# B&R Automation Studio project Panasonic_LinkaPowerCP2_A2021055 (part 5)

```iecst
(*//P4 - Spodný stoper//*)

TYPE
	P4_SpodnyStoper_typ : 	STRUCT
		IN : P4_SpodnyStoper_IN_typ;
		OUT : P4_SpodnyStoper_OUT_typ;
		PAR : P4_SpodnyStoper_PAR_typ;
		STAV : P4_SpodnyStoper_STAV_typ;
		Automat : BOOL;
		Manual : BOOL;
		Reset : BOOL;
		KoniecCyklu : BOOL;
	END_STRUCT;
	P4_SpodnyStoper_IN_typ : 	STRUCT
		PritomnostPaletky : BOOL; (*IS4_15*)
		ZaplnenieDopravnika : BOOL; (*IS4_16*)
	END_STRUCT;
	P4_SpodnyStoper_OUT_typ : 	STRUCT
		ZasunStoper : BOOL; (*YV182_VT4*)
	END_STRUCT;
	P4_SpodnyStoper_PAR_typ : 	STRUCT
		New_Member : USINT;
	END_STRUCT;
	P4_SpodnyStoper_STAV_typ : 	STRUCT
		PoINIT : BOOL;
		PrebiehaVyvezeniePaletky : BOOL;
	END_STRUCT;
END_TYPE

(*//P4 - Funkčný test A//*)

TYPE
	P4_FunkcnyTestA_typ : 	STRUCT
		CMD : P4_FunkcnyTestA_CMD_typ;
		IN : P4_FunkcnyTestA_IN_typ;
		OUT : P4_FunkcnyTestA_OUT_typ;
		PAR : P4_FunkcnyTestA_PAR_typ;
		STAV : P4_FunkcnyTestA_STAV_typ;
		RFID_hlava : SickHeads;
		Automat : BOOL;
		Manual : BOOL;
		Reset : BOOL;
		KoniecCyklu : BOOL;
	END_STRUCT;
	P4_FunkcnyTestA_CMD_typ : 	STRUCT
		RR_ZatvorTester : BOOL;
		StartTestovania : BOOL;
		RR_VysunCentrovanie : BOOL;
		RR_VysunPruzenieKontaktov : BOOL;
		OpatovnyTest : BOOL;
	END_STRUCT;
	P4_FunkcnyTestA_IN_typ : 	STRUCT
		HorneKontakty_VYSUNUTE : BOOL; (*MS4_2*)
		HorneKontakty_ZASUNUTE : BOOL; (*MS4_3*)
		SpodneKontakty_VYSUNUTE : BOOL; (*MS4_7*)
		SpodneKontakty_ZASUNUTE : BOOL; (*MS4_6*)
		Centrovanie_VYSUNUTE : BOOL; (*MS4_5*)
		Centrovanie_ZASUNUTE : BOOL; (*MS4_4*)
		TypSpodnychKontaktov_4F : BOOL;
		TypSpodnychKontaktov_5F_5H : BOOL;
	END_STRUCT;
	P4_FunkcnyTestA_OUT_typ : 	STRUCT
		ZasunStoper : BOOL; (*YV170_VT4*)
		HorneKontakty_VYSUN : BOOL; (*YV193_VT4*)
		HorneKontakty_ZASUN : BOOL; (*YV192_VT4*)
		OdpruzHornychKontaktov_VYSUN : BOOL; (*YV194_VT4*)
		OdpruzHornychKontaktov_ZASUN : BOOL; (*YV195_VT4*)
		PritlakPowerCP_VYSUN : BOOL; (*YV196_VT4*)
		SpodneKontakty_VYSUN : BOOL; (*YV200_VT4*)
		SpodneKontakty_ZASUN : BOOL; (*YV199_VT4*)
		Centrovanie_VYSUN : BOOL; (*YV197_VT4*)
		Centrovanie_ZASUN : BOOL; (*YV198_VT4*)
		KontaktyTestera_VYSUN : BOOL;
	END_STRUCT;
	P4_FunkcnyTestA_PAR_typ : 	STRUCT
		CisloPaletky_STRING : STRING[2];
		CisloPortuKlienta : UINT;
	END_STRUCT;
	P4_FunkcnyTestA_STAV_typ : 	STRUCT
		PoINIT : BOOL;
		Vysledok_FV_Testu : STRING[2]; (*OK alebo NG*)
		PrebiehaVyvezeniePaletky : BOOL;
		Tester_ON : BOOL;
		TestovanieUkoncene : BOOL;
		TesterNeodpoveda : BOOL;
		RR_SekvenciaTestera_BUSY : BOOL;
		PaletkaOznacena_NG : BOOL;
	END_STRUCT;
END_TYPE

(*//P4 - Funkčný test B//*)

TYPE
	P4_FunkcnyTestB_typ : 	STRUCT
		CMD : P4_FunkcnyTestB_CMD_typ;
		IN : P4_FunkcnyTestB_IN_typ;
		OUT : P4_FunkcnyTestB_OUT_typ;
		PAR : P4_FunkcnyTestB_PAR_typ;
		STAV : P4_FunkcnyTestB_STAV_typ;
		RFID_hlava : SickHeads;
		Automat : BOOL;
		Manual : BOOL;
		Reset : BOOL;
		KoniecCyklu : BOOL;
	END_STRUCT;
	P4_FunkcnyTestB_CMD_typ : 	STRUCT
		RR_ZatvorTester : BOOL;
		StartTestovania : BOOL;
		RR_VysunCentrovanie : BOOL;
		RR_VysunPruzenieKontaktov : BOOL;
		OpatovnyTest : BOOL;
	END_STRUCT;
	P4_FunkcnyTestB_IN_typ : 	STRUCT
		HorneKontakty_VYSUNUTE : BOOL; (*MS4_8*)
		HorneKontakty_ZASUNUTE : BOOL; (*MS4_9*)
		SpodneKontakty_VYSUNUTE : BOOL; (*MS4_13*)
		SpodneKontakty_ZASUNUTE : BOOL; (*MS4_12*)
		Centrovanie_VYSUNUTE : BOOL; (*MS4_11*)
		Centrovanie_ZASUNUTE : BOOL; (*MS4_10*)
		TypSpodnychKontaktov_4F : BOOL;
		TypSpodnychKontaktov_5F_5H : BOOL;
	END_STRUCT;
	P4_FunkcnyTestB_OUT_typ : 	STRUCT
		ZasunStoper : BOOL; (*YV171_VT4*)
		HorneKontakty_VYSUN : BOOL; (*YV202_VT4*)
		HorneKontakty_ZASUN : BOOL; (*YV201_VT4*)
		OdpruzHornychKontaktov_VYSUN : BOOL; (*YV203_VT4*)
		OdpruzHornychKontaktov_ZASUN : BOOL; (*YV204_VT4*)
		PritlakPowerCP_VYSUN : BOOL; (*YV205_VT4*)
		SpodneKontakty_VYSUN : BOOL; (*YV209_VT4*)
		SpodneKontakty_ZASUN : BOOL; (*YV208_VT4*)
		Centrovanie_VYSUN : BOOL; (*YV206_VT4*)
		Centrovanie_ZASUN : BOOL; (*YV207_VT4*)
		KontaktyTestera_VYSUN : BOOL;
	END_STRUCT;
	P4_FunkcnyTestB_PAR_typ : 	STRUCT
		CisloPaletky_STRING : STRING[2];
		CisloPortuKlienta : UINT;
	END_STRUCT;
	P4_FunkcnyTestB_STAV_typ : 	STRUCT
		PoINIT : BOOL;
		Vysledok_FV_Testu : STRING[2]; (*OK alebo NG*)
		PrebiehaVyvezeniePaletky : BOOL;
		Tester_ON : BOOL;
		TestovanieUkoncene : BOOL;
		TesterNeodpoveda : BOOL;
		RR_SekvenciaTestera_BUSY : BOOL;
		PaletkaOznacena_NG : BOOL;
	END_STRUCT;
END_TYPE

(*//P4 - Zdvižka za Funkčným Testom A//*)

TYPE
	P4_ZdvizkaZaFunkcTestA_typ : 	STRUCT
		IN : P4_ZdvizkaZaFunkTestA_IN_typ;
		OUT : P4_ZdvizkaZaFunkTestA_OUT_typ;
		PAR : P4_ZdvizkaZaFunkTestA_PAR_typ;
		STAV : P4_ZdvizkaZaFunkTestA_STAV_typ;
		Automat : BOOL;
		Manual : BOOL;
		Reset : BOOL;
		KoniecCyklu : BOOL;
	END_STRUCT;
	P4_ZdvizkaZaFunkTestA_IN_typ : 	STRUCT
		PritomnostPaletky : BOOL; (*IS4_10*)
		PoziciaPaletky_OK : BOOL; (*IS4_9*)
		Zdvizka_HornaPoloha : BOOL; (*IS4_6*)
		Zdvizka_SpodnaPoloha : BOOL; (*IS4_5*)
		Zdvizka_StrednaPoloha : BOOL; (*IS4_7*)
		TlmicPaletky_ZASUNUTY : BOOL; (*MS4_1*)
	END_STRUCT;
	P4_ZdvizkaZaFunkTestA_OUT_typ : 	STRUCT
		Zdvizku_ZASUN : BOOL; (*YV173_VT4*)
		Zdvizku_VYSUN : BOOL; (*YV172_VT4*)
		TlmicPaletky_VYSUN : BOOL; (*YV175_VT4*)
		TlmicPaletky_ZASUN : BOOL; (*YV176_VT4*)
	END_STRUCT;
	P4_ZdvizkaZaFunkTestA_PAR_typ : 	STRUCT
		New_Member : USINT;
	END_STRUCT;
	P4_ZdvizkaZaFunkTestA_STAV_typ : 	STRUCT
		PoINIT : BOOL;
		PrebiehaVyvezeniePaletky : BOOL;
	END_STRUCT;
END_TYPE

(*//P4 - Zdvižka za Funkčným Testom B//*)

TYPE
	P4_ZdvizkaZaFunkcTestB_typ : 	STRUCT
		IN : P4_ZdvizkaZaFunkTestB_IN_typ;
		OUT : P4_ZdvizkaZaFunkTestB_OUT_typ;
		PAR : P4_ZdvizkaZaFunkTestB_PAR_typ;
		STAV : P4_ZdvizkaZaFunkTestB_STAV_typ;
		Automat : BOOL;
		Manual : BOOL;
		Reset : BOOL;
		KoniecCyklu : BOOL;
	END_STRUCT;
	P4_ZdvizkaZaFunkTestB_IN_typ : 	STRUCT
		PritomnostPaletky : BOOL; (*IS4_8*)
		Zdvizka_HornaPoloha : BOOL; (*IS4_11*)
		Zdvizka_StrednaPoloha : BOOL; (*IS4_12*)
	END_STRUCT;
	P4_ZdvizkaZaFunkTestB_OUT_typ : 	STRUCT
		Zdvizku_VYSUN : BOOL; (*YV177_VT4*)
		TlmicPaletky_VYSUN : BOOL; (*YV178_VT4*)
	END_STRUCT;
	P4_ZdvizkaZaFunkTestB_PAR_typ : 	STRUCT
		New_Member : USINT;
	END_STRUCT;
	P4_ZdvizkaZaFunkTestB_STAV_typ : 	STRUCT
		PoINIT : BOOL;
		PrebiehaVyvezeniePaletky : BOOL;
	END_STRUCT;
END_TYPE

(*//P4 - Etiketovanie//*)

TYPE
	P4_Etiketovacka_typ : 	STRUCT
		CMD : P4_Etiketovacka_CMD_typ;
		IN : P4_Etiketovacka_IN_typ;
		OUT : P4_Etiketovacka_OUT_typ;
		PAR : P4_Etiketovacka_PAR_typ;
		STAV : P4_Etiketovacka_STAV_typ;
		RFID_hlava : SickHeads;
		Automat : BOOL;
		Manual : BOOL;
		Reset : BOOL;
		KoniecCyklu : BOOL;
		ServoZdvihuAplikatora : ServoDriver;
	END_STRUCT;
	P4_Etiketovacka_CMD_typ : 	STRUCT
		RR_ZdvihAplikatora_HORE : BOOL;
		RR_ZdvihAplikatora_DOLE : BOOL;
		RR_NalepEtiketu : BOOL;
		RR_VysunCentrovanie : BOOL;
		RR_PrisavanieEtikety : BOOL;
	END_STRUCT;
	P4_Etiketovacka_IN_typ : 	STRUCT
		Centrovanie_VYSUNUTE : BOOL; (*IS4_13*)
		Centrovanie_ZASUNUTE : BOOL; (*IS4_14*)
		ZdvihAplikatora_HornyLimSnimac : BOOL; (*IS4_3*)
		ZdvihAplikatora_SpodnyLimSnimac : BOOL; (*IS4_4*)
		Aplikator_OtocenyVPRED : BOOL; (*MS4_15*)
		Aplikator_OtocenyVZAD : BOOL; (*MS4_14*)
		Aplikator_VYSUNUTY : BOOL; (*MS4_17*)
		Aplikator_ZASUNUTY : BOOL; (*MS4_16*)
		PrisavanieEtikety_Vakum_OK : BOOL; (*S4_6*)
		NapajanieTlaciarne_OK : BOOL;
		PritlakPowerCP_ZASUNUTY : BOOL; (*MS4_18*)
		PritlakPowerCP_VYSUNUTY_45F : BOOL; (*MS4_19*)
		PritlakPowerCP_VYSUNUTY_5H : BOOL; (*MS4_20*)
	END_STRUCT;
	P4_Etiketovacka_OUT_typ : 	STRUCT
		OfukEtikety_ON : BOOL; (*YV185_VT4*)
		PrisavanieEtikety_ON : BOOL; (*YV210_VT4*)
		PrisavanieEtikety_OFF : BOOL; (*YV211_VT4*)
		Aplikator_OtocVPRED : BOOL; (*YV187_VT4*)
		Aplikator_OtocVZAD : BOOL; (*YV186_VT4*)
		Aplikator_VYSUN : BOOL; (*YV188_VT4*)
		ZasunStoper : BOOL; (*YV179_VT4*)
		Centrovanie_VYSUN : BOOL; (*YV180_VT4*)
		Centrovanie_ZASUN : BOOL; (*YV181_VT4*)
		PritlakPowerCP_VYSUN : BOOL; (*YV191_VT4*)
	END_STRUCT;
	P4_Etiketovacka_PAR_typ : 	STRUCT
		IndexFotky : USINT;
		CisloPaletky_STRING : STRING[2];
		ZdvihAplikatora_JoggRychlost : REAL;
		CisloPaletky : USINT;
	END_STRUCT;
	P4_Etiketovacka_STAV_typ : 	STRUCT
		PoINIT : BOOL;
		PrebiehaVyvezeniePaletky : BOOL;
		PowerCP_ZhodaQRkodu_OK : BOOL;
		Etiketa_ZhodaQRkodu_OK : BOOL;
		RR_SekvenciaEtiketovania_BUSY : BOOL;
		VstupnaKamerovaKontrola : BOOL;
		VyrobaZacala : BOOL;
	END_STRUCT;
END_TYPE

(*//P4 - Výťah*)

TYPE
	P4_Vytah_typ : 	STRUCT
		CMD : P4_Vytah_CMD_typ;
		IN : P4_Vytah_IN_typ;
		OUT : P4_Vytah_OUT_typ;
		PAR : P4_Vytah_PAR_typ;
		STAV : P4_Vytah_STAV_typ;
		Banner : BannerIOlink;
		RFID_hlava : SickHeads;
		ServoZdvihuVytahu : ServoDriver;
		Automat : BOOL;
		Manual : BOOL;
		Reset : BOOL;
		KoniecCyklu : BOOL;
	END_STRUCT;
	P4_Vytah_CMD_typ : 	STRUCT
		RR_ChodDopravnika_VPRED : BOOL;
		RR_ChodDopravnika_VZAD : BOOL;
		Banner_LED_OFF : BOOL;
		RR_ZdvihVytahu_HORE : BOOL;
		RR_ZdvihVytahu_DOLE : BOOL;
	END_STRUCT;
	P4_Vytah_IN_typ : 	STRUCT
		PrechodDopravnika : BOOL; (*OS4_1*)
		ZdvihVytahu_HornyLimitnySnimac : BOOL; (*IS4_2*)
		ZdvihVytahu_SpodnyLimitnySnimac : BOOL; (*IS4_1*)
		StavRiadeniaDopravVytahu_READY : BOOL; (*M4_3*)
		TeplotaMotoraDopravVytahu_OK : BOOL; (*M4_3*)
	END_STRUCT;
	P4_Vytah_OUT_typ : 	STRUCT
		DopravnikChod_VPRED : BOOL; (*M4_3*)
		DopravnikChod_VZAD : BOOL; (*M4_3*)
		OsvetlenieVytahu_ON : BOOL;
	END_STRUCT;
	P4_Vytah_PAR_typ : 	STRUCT
		CisloPaletky_STRING : STRING[2];
		IndexFotky : USINT;
		Zdvih_JoggRychlost : REAL;
		RR_PrecitaneCisloPaletky : USINT;
		CisloPaletky : USINT;
	END_STRUCT;
	P4_Vytah_STAV_typ : 	STRUCT
		PrebiehaVyvezeniePaletky : BOOL;
		PoINIT : BOOL;
	END_STRUCT;
END_TYPE

(**************Skrutkovacky AtlasCopco***************************)

TYPE
	SkrutkovackaAtlasCopco_typ : 	STRUCT
		RESET_Poruchy : BOOL;
		RESET_Vysledkov : BOOL;
		START_Skrutkovania : BOOL;
		START_Utahovania : BOOL;
		Stav_VysledokPotvrdeny : BOOL;
		Stav_EmergencyStop : BOOL;
		Stav_READY_to_START : BOOL;
		Stav_MANUAL : BOOL;
		Stav_UtahovanieUkoncene : BOOL;
		Stav_VysledokUtahovania_OK : BOOL;
		Stav_VysledokUtahovania_NG : BOOL;
		Stav_SmerOtacania_VPRED : BOOL;
		Stav_BUSY : BOOL;
		Stav_ControlerSwitch_ON : BOOL;
		Stav_Station_READY : BOOL;
		Stav_NastrojPripojeny : BOOL;
		Stav_NastrojUtahuje : BOOL;
		Stav_CisloAktualnehoProgramu : USINT;
		CisloZadanehoProgramu : USINT;
		VyslednyReport : STRING[5];
	END_STRUCT;
END_TYPE

(**************Ateq Leakage Testery******************)

TYPE
	AteqTester_typ : 	STRUCT
		START_Testovania : BOOL;
		RESET_Vysledkov : BOOL;
		ZMEN_Program : BOOL;
		CitajParametreTestera : BOOL;
		Stav_RESET_DONE : BOOL;
		Stav_START_DONE : BOOL;
		Stav_ZmenaProgramu_DONE : BOOL;
		Stav_ERROR : BOOL;
		Stav_READY : BOOL;
		Stav_BUSY : BOOL;
		Stav_CitanieParametrov_OK : BOOL;
		Stav_CitanieParametrov_ERROR : BOOL;
		CisloZadanehoProgramu : UINT;
		CisloAktualnehoProgramu : UINT;
		VysledokTestovania_OK : BOOL;
		VysledokTestovania_NG : BOOL;
		Profinet_PLC_INPUTS : ARRAY[1..100]OF USINT;
		Profinet_PLC_OUTPUTS : ARRAY[1..100]OF USINT;
		ReadParameter_1 : UINT;
		ReadParameter_2 : UINT;
		ReadParameter_3 : UINT;
		ReadParameter_4 : UINT;
		ReadParameter_5 : DINT;
		PocetCitanychParametrov : USINT;
		IdentifikaciaParametra_1 : USINT;
		IdentifikaciaParametra_2 : USINT;
		IdentifikaciaParametra_3 : USINT;
		IdentifikaciaParametra_4 : USINT;
		CasPnenia : REAL;
		CasStabilizacie : REAL;
		TlakPlnenia : REAL;
		Tolerancia : REAL;
		TlakUniku : REAL;
	END_STRUCT;
END_TYPE

(***************Komunikácia zo serverom********************)

TYPE
	KOM_Server_typ : 	STRUCT
		CMD : KOM_Server_CMD_typ;
		INPUTS : KOM_Server_INPUTS_typ;
		OUTPUTS : KOM_Server_OUTPUTS_typ;
		STATUS : KOM_Server_STATUS_typ;
	END_STRUCT;
	KOM_Server_CMD_typ : 	STRUCT
		VyziadajStavPaletky_TYP1 : BOOL;
		PriradQRkodFiltra_TYP3 : BOOL;
		VyziadajCisloEtikety_TYP0 : BOOL;
		OdosliStavPaletky_TYP2 : BOOL;
		VyziadajStavPanatrace_TYP4 : BOOL;
	END_STRUCT;
	KOM_Server_INPUTS_typ : 	STRUCT
		TYP_Prikazu : STRING[1]; (*Typ*)
		CisloStanice : STRING[5]; (*Stanica*)
		CisloPaletky : STRING[10]; (*RFID paletky*)
		QRkodPowerCP : STRING[30]; (*Master number*)
		QRkodFiltra : STRING[30]; (*DPS1*)
		ID_Operatora : STRING[80]; (*Operator*)
		Report : STRING[4000]; (*DATA  - Oddelené bodkočiarkou*)
		StavPaletky : STRING[4]; (*PASS alebo FAIL*)
		IndexPaletky : USINT;
	END_STRUCT;
	KOM_Server_OUTPUTS_typ : 	STRUCT
		TYP_Prikazu : STRING[1]; (*Typ*)
		CisloStanice : STRING[5]; (*Stanica*)
		CisloPaletky : STRING[10]; (*RFID paletky*)
		QRkodPowerCP : STRING[30]; (*Master number*)
		QRkodFiltra : STRING[30]; (*DPS1*)
		ID_Operatora : STRING[8]; (*Operator*)
		CisloEtikety : STRING[31];
		DruhCinnostiNaPaletke : STRING[20]; (*PRD;ST1 alebo SMP;CAL;ST1 alebo RST;HVT;ST1*)
		PovolenieCinnostiNaPaletke : STRING[2]; (*OK alebo NG*)
	END_STRUCT;
	KOM_Server_STATUS_typ : 	STRUCT
		KomunikaciaUkoncena : BOOL;
		KomunikaciaError : BOOL;
		KOM_READY : BOOL;
	END_STRUCT;
END_TYPE

(***************Vysledné reporty***************************)

TYPE
	Reports_typ : 	STRUCT
		Kamery : ReportKamery_typ;
		Skrutkovacky : ReportSkrutkovacky_typ;
		Zvaranie : ReportZvarania_typ;
		LeakageTest : ReportLeakageTest_typ;
	END_STRUCT;
	ReportKamery_typ : 	STRUCT
		P1_CAM2_KontrolaPaletky : STRING[5]; (*Výtah*)
		P1_CAM4_KontrolaPinovDPS : STRING[5]; (*Výtah*)
		P1_CAM6_KontrolaPaletky : STRING[5]; (*Srobovanie*)
		P2_CAM1_KontrolaTesnenia : STRING[5];
		P2_CAM17_KontrolaPaletky : STRING[5]; (*Zakladanie tesnenia*)
		P2_CAM9_KontrolaPaletky : STRING[5]; (*Srobovanie matice*)
		P2_CAM10_KontrolaPaletky : STRING[5]; (*Srobovanie*)
		P2_CAM11_KontrolaZvaru : STRING[5]; (*Zvaranie*)
		P2_CAM11_KontrolaPowerCP : STRING[5]; (*Zvaranie*)
		P2_CAM12_KontrolaPaletky : STRING[5];
		P3_CAM13_KontrolaPaletky : STRING[5]; (*Srobovanie*)
		P4_CAM15_KontrolaPaletky : STRING[5]; (*Etiketovačka*)
		P4_CAM16_KontrolaPaletky : STRING[5]; (*Výtah*)
	END_STRUCT;
	ReportSkrutkovacky_typ : 	STRUCT
		Moment_ToleranciaMAX : ReportSrobov_MomentTolerMAX_typ;
		Moment_ToleranciaMIN : ReportSrobov_MomentTolerMIN_typ;
		Moment_NameranaHodnota : ReportSrobov_NameranyMoment_typ;
		Uhol_ToleranciaMAX : ReportSrobov_UholTolerMAX_typ;
		Uhol_ToleranciaMIN : ReportSrobov_UholTolerMIN_typ;
		Uhol_NameranaHodnota : ReportSrobov_NameranyUhol_typ;
		VyskaSkrutkovania : ReportSrobov_VyskaSkrutkov_typ;
		CasSkrutkovania : ReportSrobov_CasSkrutkov_typ;
		VyslednyReport : ReportSrobov_VyslednyReport_typ;
	END_STRUCT;
	ReportZvarania_typ : 	STRUCT
		Vyska : ReportZvarania_Vyska_typ;
		Moment : ReportZvarania_Moment_typ;
		Frekvencia : STRING[10];
		VyslednyReport : STRING[5];
	END_STRUCT;
	ReportZvarania_Vyska_typ : 	STRUCT
		LavyZvar : STRING[10];
		PravyZvar : STRING[10];
	END_STRUCT;
	ReportZvarania_Moment_typ : 	STRUCT
		LavyZvar : STRING[4];
		PravyZvar : STRING[4];
	END_STRUCT;
	ReportSrobov_MomentTolerMAX_typ : 	STRUCT
		P1_LavaSkrutkaK30 : STRING[10];
		P1_PravaSkrutkaK30 : STRING[10];
		P1_ZadnaSkrutkaM4 : STRING[10];
		P1_PrednaSkrutkaM4 : STRING[10];
		P1_SkrutkaDPS_M4 : STRING[10];
		P1_LavaSkrutkaM5 : STRING[10];
		P1_PravaSkrutkaM5 : STRING[10];
		P1_StrednaSkrutkaM5 : STRING[10];
		P2_MaticaM4 : STRING[10];
		P2_LavaSkrutkaM6 : STRING[10];
		P2_PravaSkrutkaM6 : STRING[10];
		P2_LavaSkrutkaM4 : STRING[10];
		P2_PravaSkrutkaM4 : STRING[10];
		P2_LavaSkrutkaM5 : STRING[10];
		P2_PravaSkrutkaM5 : STRING[10];
		P2_StrednaSkrutkaM4 : STRING[10];
		P3_SkrutkaK40 : STRING[10];
		P3_SkrutkaM5 : STRING[10];
	END_STRUCT;
	ReportSrobov_MomentTolerMIN_typ : 	STRUCT
		P1_LavaSkrutkaK30 : STRING[10];
		P1_PravaSkrutkaK30 : STRING[10];
		P1_ZadnaSkrutkaM4 : STRING[10];
		P1_PrednaSkrutkaM4 : STRING[10];
		P1_SkrutkaDPS_M4 : STRING[10];
		P1_LavaSkrutkaM5 : STRING[10];
		P1_PravaSkrutkaM5 : STRING[10];
		P1_StrednaSkrutkaM5 : STRING[10];
		P2_MaticaM4 : STRING[10];
		P2_LavaSkrutkaM6 : STRING[10];
		P2_PravaSkrutkaM6 : STRING[10];
		P2_LavaSkrutkaM4 : STRING[10];
		P2_PravaSkrutkaM4 : STRING[10];
		P2_LavaSkrutkaM5 : STRING[10];
		P2_PravaSkrutkaM5 : STRING[10];
		P2_StrednaSkrutkaM4 : STRING[10];
		P3_SkrutkaK40 : STRING[10];
		P3_SkrutkaM5 : STRING[10];
	END_STRUCT;
	ReportSrobov_NameranyMoment_typ : 	STRUCT
		P1_LavaSkrutkaK30 : STRING[10];
		P1_PravaSkrutkaK30 : STRING[10];
		P1_ZadnaSkrutkaM4 : STRING[10];
		P1_PrednaSkrutkaM4 : STRING[10];
		P1_SkrutkaDPS_M4 : STRING[10];
		P1_LavaSkrutkaM5 : STRING[10];
		P1_PravaSkrutkaM5 : STRING[10];
		P1_StrednaSkrutkaM5 : STRING[10];
		P2_MaticaM4 : STRING[10];
		P2_LavaSkrutkaM6 : STRING[10];
		P2_PravaSkrutkaM6 : STRING[10];
		P2_LavaSkrutkaM4 : STRING[10];
		P2_PravaSkrutkaM4 : STRING[10];
		P2_LavaSkrutkaM5 : STRING[10];
		P2_PravaSkrutkaM5 : STRING[10];
		P2_StrednaSkrutkaM4 : STRING[10];
		P3_SkrutkaK40 : STRING[10];
		P3_SkrutkaM5 : STRING[10];
	END_STRUCT;
	ReportSrobov_UholTolerMAX_typ : 	STRUCT
		P1_LavaSkrutkaK30 : STRING[10];
		P1_PravaSkrutkaK30 : STRING[10];
		P1_ZadnaSkrutkaM4 : STRING[10];
		P1_PrednaSkrutkaM4 : STRING[10];
		P1_SkrutkaDPS_M4 : STRING[10];
		P1_LavaSkrutkaM5 : STRING[10];
		P1_PravaSkrutkaM5 : STRING[10];
		P1_StrednaSkrutkaM5 : STRING[10];
		P2_MaticaM4 : STRING[10];
		P2_LavaSkrutkaM6 : STRING[10];
		P2_PravaSkrutkaM6 : STRING[10];
		P2_LavaSkrutkaM4 : STRING[10];
		P2_PravaSkrutkaM4 : STRING[10];
		P2_LavaSkrutkaM5 : STRING[10];
		P2_PravaSkrutkaM5 : STRING[10];
		P2_StrednaSkrutkaM4 : STRING[10];
		P3_SkrutkaK40 : STRING[10];
		P3_SkrutkaM5 : STRING[10];
	END_STRUCT;
	ReportSrobov_UholTolerMIN_typ : 	STRUCT
		P1_LavaSkrutkaK30 : STRING[10];
		P1_PravaSkrutkaK30 : STRING[10];
		P1_ZadnaSkrutkaM4 : STRING[10];
		P1_PrednaSkrutkaM4 : STRING[10];
		P1_SkrutkaDPS_M4 : STRING[10];
		P1_LavaSkrutkaM5 : STRING[10];
		P1_PravaSkrutkaM5 : STRING[10];
		P1_StrednaSkrutkaM5 : STRING[10];
		P2_MaticaM4 : STRING[10];
		P2_LavaSkrutkaM6 : STRING[10];
		P2_PravaSkrutkaM6 : STRING[10];
		P2_LavaSkrutkaM4 : STRING[10];
		P2_PravaSkrutkaM4 : STRING[10];
		P2_LavaSkrutkaM5 : STRING[10];
		P2_PravaSkrutkaM5 : STRING[10];
		P2_StrednaSkrutkaM4 : STRING[10];
		P3_SkrutkaK40 : STRING[10];
		P3_SkrutkaM5 : STRING[10];
	END_STRUCT;
	ReportSrobov_NameranyUhol_typ : 	STRUCT
		P1_LavaSkrutkaK30 : STRING[10];
		P1_PravaSkrutkaK30 : STRING[10];
		P1_ZadnaSkrutkaM4 : STRING[10];
		P1_PrednaSkrutkaM4 : STRING[10];
		P1_SkrutkaDPS_M4 : STRING[10];
		P1_LavaSkrutkaM5 : STRING[10];
		P1_PravaSkrutkaM5 : STRING[10];
		P1_StrednaSkrutkaM5 : STRING[10];
		P2_MaticaM4 : STRING[10];
		P2_LavaSkrutkaM6 : STRING[10];
		P2_PravaSkrutkaM6 : STRING[10];
		P2_LavaSkrutkaM4 : STRING[10];
		P2_PravaSkrutkaM4 : STRING[10];
		P2_LavaSkrutkaM5 : STRING[10];
		P2_PravaSkrutkaM5 : STRING[10];
		P2_StrednaSkrutkaM4 : STRING[10];
		P3_SkrutkaK40 : STRING[10];
		P3_SkrutkaM5 : STRING[10];
	END_STRUCT;
	ReportSrobov_VyskaSkrutkov_typ : 	STRUCT
		P1_LavaSkrutkaK30 : STRING[10];
		P1_PravaSkrutkaK30 : STRING[10];
		P1_ZadnaSkrutkaM4 : STRING[10];
		P1_PrednaSkrutkaM4 : STRING[10];
		P1_SkrutkaDPS_M4 : STRING[10];
		P1_LavaSkrutkaM5 : STRING[10];
		P1_PravaSkrutkaM5 : STRING[10];
		P1_StrednaSkrutkaM5 : STRING[10];
		P2_MaticaM4 : STRING[10];
		P2_LavaSkrutkaM6 : STRING[10];
		P2_PravaSkrutkaM6 : STRING[10];
		P2_LavaSkrutkaM4 : STRING[10];
		P2_PravaSkrutkaM4 : STRING[10];
		P2_LavaSkrutkaM5 : STRING[10];
		P2_PravaSkrutkaM5 : STRING[10];
		P2_StrednaSkrutkaM4 : STRING[10];
		P3_SkrutkaK40 : STRING[10];
		P3_SkrutkaM5 : STRING[10];
	END_STRUCT;
	ReportSrobov_CasSkrutkov_typ : 	STRUCT
		P1_LavaSkrutkaK30 : STRING[10];
		P1_PravaSkrutkaK30 : STRING[10];
		P1_ZadnaSkrutkaM4 : STRING[10];
		P1_PrednaSkrutkaM4 : STRING[10];
		P1_SkrutkaDPS_M4 : STRING[10];
		P1_LavaSkrutkaM5 : STRING[10];
		P1_PravaSkrutkaM5 : STRING[10];
		P1_StrednaSkrutkaM5 : STRING[10];
		P2_MaticaM4 : STRING[10];
		P2_LavaSkrutkaM6 : STRING[10];
		P2_PravaSkrutkaM6 : STRING[10];
		P2_LavaSkrutkaM4 : STRING[10];
		P2_PravaSkrutkaM4 : STRING[10];
		P2_LavaSkrutkaM5 : STRING[10];
		P2_PravaSkrutkaM5 : STRING[10];
		P2_StrednaSkrutkaM4 : STRING[10];
		P3_SkrutkaK40 : STRING[10];
		P3_SkrutkaM5 : STRING[10];
	END_STRUCT;
	ReportSrobov_VyslednyReport_typ : 	STRUCT
		P1_LavaSkrutkaK30 : STRING[5];
		P1_PravaSkrutkaK30 : STRING[5];
		P1_ZadnaSkrutkaM4 : STRING[5];
		P1_PrednaSkrutkaM4 : STRING[5];
		P1_SkrutkaDPS_M4 : STRING[5];
		P1_LavaSkrutkaM5 : STRING[5];
		P1_PravaSkrutkaM5 : STRING[5];
		P1_StrednaSkrutkaM5 : STRING[5];
		P2_MaticaM4 : STRING[5];
		P2_LavaSkrutkaM6 : STRING[5];
		P2_PravaSkrutkaM6 : STRING[5];
		P2_LavaSkrutkaM4 : STRING[5];
		P2_PravaSkrutkaM4 : STRING[5];
		P2_LavaSkrutkaM5 : STRING[5];
		P2_PravaSkrutkaM5 : STRING[5];
		P2_StrednaSkrutkaM4 : STRING[5];
		P3_SkrutkaK40 : STRING[5];
		P3_SkrutkaM5 : STRING[5];
	END_STRUCT;
	ReportLeakageTest_typ : 	STRUCT
		CasPlnenia : RepLeakTest_CasPlnenia_typ;
		CasStabilizacie : RepLeakTest_CasStabilizacie_typ;
		TlakPlnenia : RepLeakTest_TlakPlnenia_typ;
		TlakPritlaku : RepLeakTest_TlakPritlaku_typ;
		ToleranciaPritlaku_MIN : RepLeakTest_TolPritlakuMIN_typ;
		ToleranciaPritlaku_MAX : RepLeakTest_TolPritlakuMAX_typ;
		ToleranciaTlakUniku_MIN : RepLeakTest_TolTlakUnikuMIN_typ;
		ToleranciaTlakUniku_MAX : RepLeakTest_TolTlakUnikuMAX_typ;
		TlakUniku : RepLeakTest_TlakUniku_typ;
		Tolerancia : RepLeakTest_Tolerancia_typ;
		VyslednyReport : RepLeakTest_VyslednyReport_typ;
	END_STRUCT;
	RepLeakTest_CasPlnenia_typ : 	STRUCT
		StanicaA : STRING[10];
		StanicaB : STRING[10];
	END_STRUCT;
	RepLeakTest_CasStabilizacie_typ : 	STRUCT
		StanicaA : STRING[10];
		StanicaB : STRING[10];
	END_STRUCT;
	RepLeakTest_TlakPlnenia_typ : 	STRUCT
		StanicaA : STRING[10];
		StanicaB : STRING[10];
	END_STRUCT;
	RepLeakTest_TlakPritlaku_typ : 	STRUCT
		StanicaA : STRING[10];
		StanicaB : STRING[10];
	END_STRUCT;
	RepLeakTest_TolPritlakuMIN_typ : 	STRUCT
		StanicaA : STRING[10];
		StanicaB : STRING[10];
	END_STRUCT;
	RepLeakTest_TolPritlakuMAX_typ : 	STRUCT
		StanicaA : STRING[10];
		StanicaB : STRING[10];
	END_STRUCT;
	RepLeakTest_TlakUniku_typ : 	STRUCT
		StanicaA : STRING[10];
		StanicaB : STRING[10];
	END_STRUCT;
	RepLeakTest_TolTlakUnikuMIN_typ : 	STRUCT
		StanicaA : STRING[10];
		StanicaB : STRING[10];
	END_STRUCT;
	RepLeakTest_TolTlakUnikuMAX_typ : 	STRUCT
		StanicaA : STRING[10];
		StanicaB : STRING[10];
	END_STRUCT;
	RepLeakTest_Tolerancia_typ : 	STRUCT
		StanicaA : STRING[10];
		StanicaB : STRING[10];
	END_STRUCT;
	RepLeakTest_VyslednyReport_typ : 	STRUCT
		StanicaA : STRING[5];
		StanicaB : STRING[5];
	END_STRUCT;
END_TYPE

(****************Kamerove kontroly**************************)

TYPE
	CAM1_typ : 	STRUCT  (*P2_ST1_ZaklTesnenia - Kontrola tesnenia a QR kódu Power CP //CAM4//*)
		CMD : CAM1_Commands_typ;
		PAR : CAM1_Parametre_typ;
		STAV : CAM1_Status_typ;
		RESULT : CAM1_Results_typ;
		Profinet_PLC_INPUTS : ARRAY[0..100]OF USINT;
		Profinet_PLC_OUTPUTS : ARRAY[0..3]OF USINT;
	END_STRUCT;
	CAM1_Commands_typ : 	STRUCT
		Triger : BOOL;
		OdosliFotku : BOOL;
		VymazFotku : BOOL;
	END_STRUCT;
	CAM1_Parametre_typ : 	STRUCT
		ResultFotky : STRING[5];
	END_STRUCT;
	CAM1_Status_typ : 	STRUCT
		BUSY : BOOL;
		SWITCH : BOOL;
		READY : BOOL;
		OLD_SWITCH : BOOL;
		Results_READY : BOOL;
		Command_READY : BOOL;
		Command_ERROR : BOOL;
		Command_AKCEPTOVANY : BOOL;
		RunCounter : UINT;
		OldRunCounter : UINT;
		RunCounter_Byte0 : USINT;
		RunCounter_Byte1 : USINT;
	END_STRUCT;
	CAM1_Results_typ : 	STRUCT
		ZalozenieTesnenia_OK : BOOL;
		NepritomnostTesnenia : BOOL;
	END_STRUCT;
	CAM2_typ : 	STRUCT  (*P1_ST1_Vytah - kontrola kusov na paletke //CAM1//*)
		CMD : CAM2_Commands_typ;
		PAR : CAM2_Parametre_typ;
		STAV : CAM2_Status_typ;
		RESULT : CAM2_Results_typ;
		Profinet_PLC_INPUTS : ARRAY[0..100]OF USINT;
		Profinet_PLC_OUTPUTS : ARRAY[0..3]OF USINT;
	END_STRUCT;
	CAM2_Commands_typ : 	STRUCT
		Triger : BOOL;
		OdosliFotku : BOOL;
		VymazFotku : BOOL;
	END_STRUCT;
	CAM2_Parametre_typ : 	STRUCT
		ResultFotky : STRING[5];
	END_STRUCT;
	CAM2_Status_typ : 	STRUCT
		READY : BOOL;
		BUSY : BOOL;
		SWITCH : BOOL;
		OLD_SWITCH : BOOL;
		Results_READY : BOOL;
		Command_READY : BOOL;
		Command_ERROR : BOOL;
		Command_AKCEPTOVANY : BOOL;
		RunCounter : UINT;
		OldRunCounter : UINT;
		RunCounter_Byte0 : USINT;
		RunCounter_Byte1 : USINT;
	END_STRUCT;
	CAM2_Results_typ : 	STRUCT
		Paletka : CAM2_Paletka_typ;
		PowerCP : CAM2_PowerCP_typ;
	END_STRUCT;
	CAM2_PowerCP_typ : 	STRUCT
		New_Member : USINT;
	END_STRUCT;
	CAM2_Paletka_typ : 	STRUCT
		Pritom_PowerCP_5F : BOOL;
		Pritom_PowerCP_4F : BOOL;
		Pritom_PowerCP_5H : BOOL;
		Pritomn_Skeletonu_5H : BOOL;
		Pritomn_Skeletonu_4F5F : BOOL;
		Pritom_Busbarov_Spodne_5H : BOOL;
		Pritom_Busbaru_Spodny_5F : BOOL;
		Pritom_Busbaru_Spodny_4F : BOOL;
		Pritom_DPS_4F5F : BOOL;
		Pritom_Foamu_Lavy_4F5F : BOOL;
		Pritom_Foamu_Pravy_4F5F : BOOL;
	END_STRUCT;
	CAM3_typ : 	STRUCT  (*P1_ST1_Vytah - kontrola QR kódu DPS //Smart kamera//*)
		CMD : CAM3_Commands_typ;
		PAR : CAM3_Parametre_typ;
		STAV : CAM3_Status_typ;
		RESULT : CAM3_Results_typ;
		Profinet_QRkod_Znaky : ARRAY[0..31]OF USINT;
		Profinet_PLC_INPUTS : ARRAY[0..100]OF USINT;
		Profinet_PLC_OUTPUTS : ARRAY[0..3]OF USINT;
	END_STRUCT;
	CAM3_Commands_typ : 	STRUCT
		Triger : BOOL;
		OdosliFotku : BOOL;
		VymazFotku : BOOL;
	END_STRUCT;
	CAM3_Parametre_typ : 	STRUCT
		ResultFotky : STRING[5];
	END_STRUCT;
	CAM3_Status_typ : 	STRUCT
		BUSY : BOOL;
		SWITCH : BOOL;
		READY : BOOL;
		OLD_SWITCH : BOOL;
		Results_READY : BOOL;
		RunCounter : UINT;
		OldRunCounter : UINT;
		RunCounter_Byte0 : USINT;
		RunCounter_Byte1 : USINT;
	END_STRUCT;
	CAM3_Results_typ : 	STRUCT
		Paletka : CAM3_Paletka_typ;
		PowerCP : CAM3_PowerCP_typ;
	END_STRUCT;
	CAM3_PowerCP_typ : 	STRUCT
		New_Member : USINT;
	END_STRUCT;
	CAM3_Paletka_typ : 	STRUCT
		CitanieQRkodu_DPS_OK : BOOL;
		PrecitanyQRkod_DPS : STRING[32];
	END_STRUCT;
	CAM4_typ : 	STRUCT  (*P1_ST1_Vytah - kontrola klipov krytu DPS //CAM2//*)
		CMD : CAM4_Commands_typ;
		PAR : CAM4_Parametre_typ;
		STAV : CAM4_Status_typ;
		RESULT : CAM4_Results_typ;
		Profinet_PLC_INPUTS : ARRAY[0..100]OF USINT;
		Profinet_PLC_OUTPUTS : ARRAY[0..3]OF USINT;
	END_STRUCT;
	CAM4_Commands_typ : 	STRUCT
		Triger : BOOL;
		OdosliFotku : BOOL;
		VymazFotku : BOOL;
	END_STRUCT;
	CAM4_Parametre_typ : 	STRUCT
		ResultFotky : STRING[5];
	END_STRUCT;
	CAM4_Status_typ : 	STRUCT
		READY : BOOL;
		BUSY : BOOL;
		SWITCH : BOOL;
		OLD_SWITCH : BOOL;
		Results_READY : BOOL;
		Command_READY : BOOL;
		Command_ERROR : BOOL;
		Command_AKCEPTOVANY : BOOL;
		RunCounter : UINT;
		OldRunCounter : UINT;
		RunCounter_Byte0 : USINT;
		RunCounter_Byte1 : USINT;
	END_STRUCT;
	CAM4_Results_typ : 	STRUCT
		Paletka : CAM4_Paletka_typ;
		PowerCP : CAM4_PowerCP_typ;
	END_STRUCT;
	CAM4_PowerCP_typ : 	STRUCT
		New_Member : USINT;
	END_STRUCT;
	CAM4_Paletka_typ : 	STRUCT
		Pritomn_Pinu1_KrytDPS_4F5F : BOOL;
		Pritomn_Pinu2_KrytDPS_4F5F : BOOL;
		Pritomn_Pinu3_KrytDPS_4F5F : BOOL;
		Pritomn_Pinu4_KrytDPS_4F5F : BOOL;
		Pritomn_Pinu5_KrytDPS_4F5F : BOOL;
		Pritomn_Pinu6_KrytDPS_4F5F : BOOL;
		Pritom_DPS_4F5F : BOOL;
	END_STRUCT;
	CAM5_typ : 	STRUCT  (*P1_ST1_Vytah - kontrola QR kódu PowerCP//Smart kamera//*)
		CMD : CAM5_Commands_typ;
		PAR : CAM5_Parametre_typ;
		STAV : CAM5_Status_typ;
		RESULT : CAM5_Results_typ;
		Profinet_QRkod_Znaky : ARRAY[0..31]OF USINT;
		Profinet_PLC_INPUTS : ARRAY[0..100]OF USINT;
		Profinet_PLC_OUTPUTS : ARRAY[0..3]OF USINT;
	END_STRUCT;
	CAM5_Commands_typ : 	STRUCT
		Triger : BOOL;
		OdosliFotku : BOOL;
		VymazFotku : BOOL;
	END_STRUCT;
	CAM5_Parametre_typ : 	STRUCT
		ResultFotky : STRING[5];
	END_STRUCT;
	CAM5_Status_typ : 	STRUCT
		BUSY : BOOL;
		SWITCH : BOOL;
		READY : BOOL;
		OLD_SWITCH : BOOL;
		Results_READY : BOOL;
		RunCounter : UINT;
		OldRunCounter : UINT;
		RunCounter_Byte0 : USINT;
		RunCounter_Byte1 : USINT;
	END_STRUCT;
	CAM5_Results_typ : 	STRUCT
		Paletka : CAM5_Paletka_typ;
		PowerCP : CAM5_PowerCP_typ;
	END_STRUCT;
	CAM5_PowerCP_typ : 	STRUCT
		CitanieQRkodu_PowerCP_OK : BOOL;
		PrecitanyQRkod_PowerCP : STRING[32];
	END_STRUCT;
	CAM5_Paletka_typ : 	STRUCT
		New_Member : USINT;
	END_STRUCT;
	CAM6_typ : 	STRUCT  (*P1_ST2_StoperSkrutkovania - Kontrola paletky //CAM3//*)
		CMD : CAM6_Commands_typ;
		PAR : CAM6_Parametre_typ;
		STAV : CAM6_Status_typ;
		RESULT : CAM6_Results_typ;
		Profinet_PLC_INPUTS : ARRAY[0..100]OF USINT;
		Profinet_PLC_OUTPUTS : ARRAY[0..3]OF USINT;
	END_STRUCT;
	CAM6_Commands_typ : 	STRUCT
		Triger : BOOL;
		OdosliFotku : BOOL;
		VymazFotku : BOOL;
	END_STRUCT;
	CAM6_Parametre_typ : 	STRUCT
		ResultFotky : STRING[5];
	END_STRUCT;
	CAM6_Status_typ : 	STRUCT
		READY : BOOL;
		BUSY : BOOL;
		SWITCH : BOOL;
		OLD_SWITCH : BOOL;
		Results_READY : BOOL;
		Command_READY : BOOL;
		Command_ERROR : BOOL;
		Command_AKCEPTOVANY : BOOL;
		RunCounter : UINT;
		OldRunCounter : UINT;
		RunCounter_Byte0 : USINT;
		RunCounter_Byte1 : USINT;
	END_STRUCT;
	CAM6_Results_typ : 	STRUCT
		Paletka : CAM6_Paletka_typ;
		PowerCP : CAM6_PowerCP_typ;
	END_STRUCT;
	CAM6_PowerCP_typ : 	STRUCT
		Nepritom_LavyFoam_4F5F : BOOL;
		Nepritom_PravyFoam_4F5F : BOOL;
		Pritom_LavejSkrutkyK30 : BOOL;
		Pritom_PravejSkrutkyK30 : BOOL;
	END_STRUCT;
	CAM6_Paletka_typ : 	STRUCT
		Pritom_PowerCP_5H : BOOL;
		Pritom_PowerCP_4F : BOOL;
		Pritom_PowerCP_5F : BOOL;
		Pritom_DPS_45F : BOOL;
		Pritom_SpodnychBusbarov_5H : BOOL;
		Pritom_SpodnyBusbar_5F : BOOL;
		Pritom_SpodnyBusbar_4F : BOOL;
		Pritom_LavyFoam_4F5F : BOOL;
		Pritom_PravyFoam_4F5F : BOOL;
	END_STRUCT;
	CAM7_typ : 	STRUCT  (*P2_ST1_StoperZaklTesnenia - Kontrola Power CP a QR kódu filtra //CAM5//*)
		CMD : CAM7_Commands_typ;
		PAR : CAM7_Parametre_typ;
		STAV : CAM7_Status_typ;
		RESULT : CAM7_Results_typ;
		Profinet_QRkod_Znaky : ARRAY[0..31]OF USINT;
		Profinet_PLC_INPUTS : ARRAY[0..100]OF USINT;
		Profinet_PLC_OUTPUTS : ARRAY[0..3]OF USINT;
	END_STRUCT;
	CAM7_Commands_typ : 	STRUCT
		Triger : BOOL;
		OdosliFotku : BOOL;
		VymazFotku : BOOL;
	END_STRUCT;
	CAM7_Parametre_typ : 	STRUCT
		ResultFotky : STRING[5];
	END_STRUCT;
	CAM7_Status_typ : 	STRUCT
		BUSY : BOOL;
		SWITCH : BOOL;
		READY : BOOL;
		OLD_SWITCH : BOOL;
		Results_READY : BOOL;
		Command_READY : BOOL;
		Command_ERROR : BOOL;
		Command_AKCEPTOVANY : BOOL;
		RunCounter : UINT;
		OldRunCounter : UINT;
		RunCounter_Byte0 : USINT;
		RunCounter_Byte1 : USINT;
	END_STRUCT;
	CAM7_Results_typ : 	STRUCT
		CitanieQRkodu_Filtra5H_OK : BOOL;
		PrecitanyQRkod_Filtra5H : STRING[32];
	END_STRUCT;
	CAM8_typ : 	STRUCT  (*P2_ST1_StoperZaklTesnenia - Kontrola spodného QR kódu Power CP //Smart kamera//*)
		CMD : CAM8_Commands_typ;
		PAR : CAM8_Parametre_typ;
		STAV : CAM8_Status_typ;
		RESULT : CAM8_Results_typ;
		Profinet_QRkod_Znaky : ARRAY[0..31]OF USINT;
		Profinet_PLC_INPUTS : ARRAY[0..100]OF USINT;
		Profinet_PLC_OUTPUTS : ARRAY[0..3]OF USINT;
	END_STRUCT;
	CAM8_Commands_typ : 	STRUCT
		Triger : BOOL;
		OdosliFotku : BOOL;
		VymazFotku : BOOL;
	END_STRUCT;
	CAM8_Parametre_typ : 	STRUCT
		ResultFotky : STRING[5];
	END_STRUCT;
	CAM8_Status_typ : 	STRUCT
		BUSY : BOOL;
		SWITCH : BOOL;
		READY : BOOL;
		OLD_SWITCH : BOOL;
		Results_READY : BOOL;
		RunCounter : UINT;
		OldRunCounter : UINT;
		RunCounter_Byte0 : USINT;
		RunCounter_Byte1 : USINT;
	END_STRUCT;
	CAM8_Results_typ : 	STRUCT
		Paletka : CAM8_Paletka_typ;
		PowerCP : CAM8_PowerCP_typ;
	END_STRUCT;
	CAM8_PowerCP_typ : 	STRUCT
		CitanieQRkodu_PowerCP_OK : BOOL;
		PrecitanyQRkod_PowerCP : STRING[30];
	END_STRUCT;
	CAM8_Paletka_typ : 	STRUCT
		New_Member : USINT;
	END_STRUCT;
	CAM9_typ : 	STRUCT  (*P2_ST2_StoperMaticovacky - Kontrola paletky //Smart kamera//*)
		CMD : CAM9_Commands_typ;
		PAR : CAM9_Parametre_typ;
		STAV : CAM9_Status_typ;
		RESULT : CAM9_Results_typ;
		Profinet_PLC_INPUTS : ARRAY[0..100]OF USINT;
		Profinet_PLC_OUTPUTS : ARRAY[0..3]OF USINT;
	END_STRUCT;
	CAM9_Commands_typ : 	STRUCT
		Triger : BOOL;
		OdosliFotku : BOOL;
		VymazFotku : BOOL;
	END_STRUCT;
	CAM9_Parametre_typ : 	STRUCT
		ResultFotky : STRING[5];
	END_STRUCT;
	CAM9_Status_typ : 	STRUCT
		BUSY : BOOL;
		SWITCH : BOOL;
		READY : BOOL;
		OLD_SWITCH : BOOL;
		Results_READY : BOOL;
		RunCounter : UINT;
		OldRunCounter : UINT;
		RunCounter_Byte0 : USINT;
		RunCounter_Byte1 : USINT;
	END_STRUCT;
	CAM9_Results_typ : 	STRUCT
		Paletka : CAM9_Paletka_typ;
		PowerCP : CAM9_PowerCP_typ;
	END_STRUCT;
	CAM9_PowerCP_typ : 	STRUCT
		PritomMatice : BOOL;
		PritomnBusbaru_5H : BOOL;
	END_STRUCT;
	CAM9_Paletka_typ : 	STRUCT
		New_Member : USINT;
	END_STRUCT;
	CAM10_typ : 	STRUCT  (*P2_ST3_StoperSkrutkovania - Kontrola paletky //CAM7//*)
		CMD : CAM10_Commands_typ;
		PAR : CAM10_Parametre_typ;
		STAV : CAM10_Status_typ;
		RESULT : CAM10_Results_typ;
		Profinet_PLC_INPUTS : ARRAY[0..100]OF USINT;
		Profinet_PLC_OUTPUTS : ARRAY[0..3]OF USINT;
	END_STRUCT;
	CAM10_Commands_typ : 	STRUCT
		Triger : BOOL;
		OdosliFotku : BOOL;
		VymazFotku : BOOL;
	END_STRUCT;
	CAM10_Parametre_typ : 	STRUCT
		ResultFotky : STRING[5];
	END_STRUCT;
	CAM10_Status_typ : 	STRUCT
		BUSY : BOOL;
		SWITCH : BOOL;
		READY : BOOL;
		OLD_SWITCH : BOOL;
		Results_READY : BOOL;
		Command_READY : BOOL;
		Command_ERROR : BOOL;
		Command_AKCEPTOVANY : BOOL;
		RunCounter : UINT;
		OldRunCounter : UINT;
		RunCounter_Byte0 : USINT;
		RunCounter_Byte1 : USINT;
	END_STRUCT;
	CAM10_Results_typ : 	STRUCT
		Paletka : CAM10_Paletka_typ;
		PowerCP : CAM10_PowerCP_typ;
	END_STRUCT;
	CAM10_PowerCP_typ : 	STRUCT
		New_Member : USINT;
	END_STRUCT;
	CAM10_Paletka_typ : 	STRUCT
		Pritomn_Busbarov_45F : BOOL;
		Pritomn_Busbarov_5H : BOOL;
		Pritomn_PowerCP_5H : BOOL;
		Pritomn_PowerCP_4F : BOOL;
		Pritomn_PowerCP_5F : BOOL;
	END_STRUCT;
	CAM11_typ : 	STRUCT  (*P2_ST4_StoperZvarania - Kontrola pravého MV case //CAM8//*)
		CMD : CAM11_Commands_typ;
		PAR : CAM11_Parametre_typ;
		STAV : CAM11_Status_typ;
		RESULT : CAM11_Results_typ;
		Profinet_PLC_INPUTS : ARRAY[0..100]OF USINT;
		Profinet_PLC_OUTPUTS : ARRAY[0..3]OF USINT;
	END_STRUCT;
	CAM11_Commands_typ : 	STRUCT
		Triger : BOOL;
		OdosliFotku : BOOL;
		VymazFotku : BOOL;
	END_STRUCT;
	CAM11_Parametre_typ : 	STRUCT
		ResultFotky : STRING[5];
	END_STRUCT;
	CAM11_Status_typ : 	STRUCT
		BUSY : BOOL;
		SWITCH : BOOL;
		READY : BOOL;
		OLD_SWITCH : BOOL;
		Results_READY : BOOL;
		Command_READY : BOOL;
		Command_ERROR : BOOL;
		Command_AKCEPTOVANY : BOOL;
		RunCounter : UINT;
		OldRunCounter : UINT;
		RunCounter_Byte0 : USINT;
		RunCounter_Byte1 : USINT;
	END_STRUCT;
	CAM11_Results_typ : 	STRUCT
		Paletka : CAM11_Paletka_typ;
		PowerCP : CAM11_PowerCP_typ;
	END_STRUCT;
	CAM11_Paletka_typ : 	STRUCT
		Pritomn_PowerCP_4F : BOOL;
		Pritomn_PowerCP_5F : BOOL;
		Pritomn_PowerCP_5H : BOOL;
	END_STRUCT;
	CAM11_PowerCP_typ : 	STRUCT
		Pritomn_LavyMVcase : BOOL;
		Pritomn_PravyMVcase : BOOL;
		LavyBusbar_Zvaranie_OK : BOOL;
		PravyBusbar_Zvaranie_OK : BOOL;
		Pritomn_TopCover_4F : BOOL;
		Pritomn_TopCover_5F : BOOL;
		Pritomn_TopCover_5H : BOOL;
	END_STRUCT;
	CAM12_typ : 	STRUCT  (*P2_ST4_StoperZvarania - Kontrola lavého MV case a Power CP //CAM9//*)
		CMD : CAM12_Commands_typ;
		PAR : CAM12_Parametre_typ;
		STAV : CAM12_Status_typ;
		RESULT : CAM12_Results_typ;
		Profinet_PLC_INPUTS : ARRAY[0..100]OF USINT;
		Profinet_PLC_OUTPUTS : ARRAY[0..3]OF USINT;
	END_STRUCT;
	CAM12_Commands_typ : 	STRUCT
		Triger : BOOL;
		OdosliFotku : BOOL;
		VymazFotku : BOOL;
	END_STRUCT;
	CAM12_Parametre_typ : 	STRUCT
		ResultFotky : STRING[5];
	END_STRUCT;
	CAM12_Status_typ : 	STRUCT
		BUSY : BOOL;
		SWITCH : BOOL;
		READY : BOOL;
		OLD_SWITCH : BOOL;
		Results_READY : BOOL;
		Command_READY : BOOL;
		Command_ERROR : BOOL;
		Command_AKCEPTOVANY : BOOL;
		RunCounter : UINT;
		OldRunCounter : UINT;
		RunCounter_Byte0 : USINT;
		RunCounter_Byte1 : USINT;
	END_STRUCT;
	CAM12_Results_typ : 	STRUCT
		Paletka : CAM12_Paletka_typ;
		PowerCP : CAM12_PowerCP_typ;
	END_STRUCT;
	CAM12_Paletka_typ : 	STRUCT
		Pritomn_TopCover_5H : BOOL;
		Pritomn_TopCover_4F : BOOL;
		Pritomn_TopCover_5F : BOOL;
		Pritomn_LavyMVcase : BOOL;
		Pritomn_PravyMVcase : BOOL;
	END_STRUCT;
	CAM12_PowerCP_typ : 	STRUCT
		New_Member : USINT;
	END_STRUCT;
	CAM13_typ : 	STRUCT  (*P3_ST1_StoperSkrutkovania - Kontrola paletky //Kamerová kontrola zrušená//*)
		CMD : CAM13_Commands_typ;
		PAR : CAM13_Parametre_typ;
		STAV : CAM13_Status_typ;
		RESULT : CAM13_Results_typ;
		Profinet_PLC_INPUTS : ARRAY[0..100]OF USINT;
		Profinet_PLC_OUTPUTS : ARRAY[0..3]OF USINT;
	END_STRUCT;
	CAM13_Commands_typ : 	STRUCT
		Triger : BOOL;
		OdosliFotku : BOOL;
		VymazFotku : BOOL;
	END_STRUCT;
	CAM13_Parametre_typ : 	STRUCT
		ResultFotky : STRING[5];
	END_STRUCT;
	CAM13_Status_typ : 	STRUCT
		BUSY : BOOL;
		SWITCH : BOOL;
		READY : BOOL;
		OLD_SWITCH : BOOL;
		Results_READY : BOOL;
		Command_READY : BOOL;
		Command_ERROR : BOOL;
		Command_AKCEPTOVANY : BOOL;
		RunCounter : UINT;
		OldRunCounter : UINT;
		RunCounter_Byte0 : USINT;
		RunCounter_Byte1 : USINT;
	END_STRUCT;
	CAM13_Results_typ : 	STRUCT
		Pritomn_SkrutkyK40_TopCover_4F5F : BOOL;
		Pritomn_SkrutkyM5_TopCover : BOOL;
	END_STRUCT;
	CAM14_typ : 	STRUCT  (*P4_ST3_StoperEtiketovania - kontrola QR kodu na Power CP //Smart kamera//*)
		CMD : CAM14_Commands_typ;
		PAR : CAM14_Parametre_typ;
		STAV : CAM14_Status_typ;
		RESULT : CAM14_Results_typ;
		Profinet_QRkod_Znaky : ARRAY[0..31]OF USINT;
		Profinet_PLC_INPUTS : ARRAY[0..100]OF USINT;
		Profinet_PLC_OUTPUTS : ARRAY[0..3]OF USINT;
	END_STRUCT;
	CAM14_Commands_typ : 	STRUCT
		Triger : BOOL;
		OdosliFotku : BOOL;
		VymazFotku : BOOL;
	END_STRUCT;
	CAM14_Parametre_typ : 	STRUCT
		ResultFotky : STRING[5];
	END_STRUCT;
	CAM14_Status_typ : 	STRUCT
		BUSY : BOOL;
		SWITCH : BOOL;
		READY : BOOL;
		OLD_SWITCH : BOOL;
		Results_READY : BOOL;
		RunCounter : UINT;
		OldRunCounter : UINT;
		RunCounter_Byte0 : USINT;
		RunCounter_Byte1 : USINT;
	END_STRUCT;
	CAM14_Results_typ : 	STRUCT
		Paletka : CAM14_Paletka_typ;
		PowerCP : CAM14_PowerCP_typ;
	END_STRUCT;
	CAM14_PowerCP_typ : 	STRUCT
		CitanieQRkodu_PowerCP_OK : BOOL;
		PrecitanyQRkod_PowerCP : STRING[32];
	END_STRUCT;
	CAM14_Paletka_typ : 	STRUCT
		New_Member : USINT;
	END_STRUCT;
	CAM15_typ : 	STRUCT  (*P4_ST3_StoperEtiketovania - kontrola nalepenej etikety //CAM10//*)
		CMD : CAM15_Commands_typ;
		PAR : CAM15_Parametre_typ;
		STAV : CAM15_Status_typ;
		RESULT : CAM15_Results_typ;
		Profinet_QRkod_Znaky : ARRAY[0..31]OF USINT;
		Profinet_PLC_INPUTS : ARRAY[0..100]OF USINT;
		Profinet_PLC_OUTPUTS : ARRAY[0..3]OF USINT;
	END_STRUCT;
	CAM15_Commands_typ : 	STRUCT
		Triger : BOOL;
		OdosliFotku : BOOL;
		VymazFotku : BOOL;
	END_STRUCT;
	CAM15_Parametre_typ : 	STRUCT
		ResultFotky : STRING[5];
	END_STRUCT;
	CAM15_Status_typ : 	STRUCT
		BUSY : BOOL;
		SWITCH : BOOL;
		READY : BOOL;
		OLD_SWITCH : BOOL;
		Results_READY : BOOL;
		Command_READY : BOOL;
		Command_ERROR : BOOL;
		Command_AKCEPTOVANY : BOOL;
		RunCounter : UINT;
		OldRunCounter : UINT;
		RunCounter_Byte0 : USINT;
		RunCounter_Byte1 : USINT;
	END_STRUCT;
	CAM15_Results_typ : 	STRUCT
		Pritomn_Etikety : BOOL;
		Pritomn_LogoBMV : BOOL;
		Pritomn_LogoPanasonic : BOOL;
		CitanieQRkodu_Etikety_OK : BOOL;
		PrecitanyQRkod_Etikety : STRING[31];
	END_STRUCT;
	CAM16_typ : 	STRUCT  (*P4_ST4_Vytah - kontrola paletky //CAM11//*)
		CMD : CAM16_Commands_typ;
		PAR : CAM16_Parametre_typ;
		STAV : CAM16_Status_typ;
		RESULT : CAM16_Results_typ;
		Profinet_PLC_INPUTS : ARRAY[0..100]OF USINT;
		Profinet_PLC_OUTPUTS : ARRAY[0..3]OF USINT;
	END_STRUCT;
	CAM16_Commands_typ : 	STRUCT
		Triger : BOOL;
		OdosliFotku : BOOL;
		VymazFotku : BOOL;
	END_STRUCT;
	CAM16_Parametre_typ : 	STRUCT
		ResultFotky : STRING[5];
	END_STRUCT;
	CAM16_Status_typ : 	STRUCT
		BUSY : BOOL;
		SWITCH : BOOL;
		READY : BOOL;
		OLD_SWITCH : BOOL;
		Results_READY : BOOL;
		Command_READY : BOOL;
		Command_ERROR : BOOL;
		Command_AKCEPTOVANY : BOOL;
		RunCounter : UINT;
		OldRunCounter : UINT;
		RunCounter_Byte0 : USINT;
		RunCounter_Byte1 : USINT;
	END_STRUCT;
	CAM16_Results_typ : 	STRUCT
		New_Member : USINT;
		Paletka : CAM16_Paletka_typ;
		PowerCP : CAM16_PowerCP_typ;
	END_STRUCT;
	CAM16_Paletka_typ : 	STRUCT
		Pritomn_Busbarov_4F : BOOL;
		Pritomn_Busbarov_5F : BOOL;
		Pritomn_Busbarov_5H : BOOL;
		Pritomn_LavyMVcase : BOOL;
		Pritomn_PravyMVcase : BOOL;
		Pritomn_PowerCP : BOOL;
		PrazdnaPaletka : BOOL;
	END_STRUCT;
	CAM16_PowerCP_typ : 	STRUCT
		New_Member : USINT;
	END_STRUCT;
	CAM17_typ : 	STRUCT  (*P2_ST1_StoperZaklTesnenia - Kontrola paletky //CAM6//*)
		CMD : CAM17_Commands_typ;
		PAR : CAM17_Parametre_typ;
		STAV : CAM17_Status_typ;
		RESULT : CAM17_Results_typ;
		Profinet_QRkod_Znaky : ARRAY[0..31]OF USINT;
		Profinet_PLC_INPUTS : ARRAY[0..100]OF USINT;
		Profinet_PLC_OUTPUTS : ARRAY[0..3]OF USINT;
	END_STRUCT;
	CAM17_Commands_typ : 	STRUCT
		Triger : BOOL;
		OdosliFotku : BOOL;
		VymazFotku : BOOL;
	END_STRUCT;
	CAM17_Parametre_typ : 	STRUCT
		ResultFotky : STRING[5];
	END_STRUCT;
	CAM17_Status_typ : 	STRUCT
		BUSY : BOOL;
		SWITCH : BOOL;
		READY : BOOL;
		OLD_SWITCH : BOOL;
		Results_READY : BOOL;
		Command_READY : BOOL;
		Command_ERROR : BOOL;
		Command_AKCEPTOVANY : BOOL;
		RunCounter : UINT;
		OldRunCounter : UINT;
		RunCounter_Byte0 : USINT;
		RunCounter_Byte1 : USINT;
	END_STRUCT;
	CAM17_Results_typ : 	STRUCT
		Paletka : CAM17_Paletka_typ;
		PowerCP : CAM17_PowerCP_typ;
	END_STRUCT;
	CAM17_PowerCP_typ : 	STRUCT
		New_Member : USINT;
	END_STRUCT;
	CAM17_Paletka_typ : 	STRUCT
		Pritomn_TopCoveru_4F : BOOL;
		Pritomn_TopCoveru_5F : BOOL;
		Pritomn_TopCoveru_5H : BOOL;
		Pritomn_Busbary_5H : BOOL;
		Pritomn_Busbary_5F : BOOL;
		Pritomn_Busbary_4F : BOOL;
		Pritomn_LavyMVcase : BOOL;
		Pritomn_PravyMVcase : BOOL;
		Pritomn_PowerCP_4F : BOOL;
		Pritomn_PowerCP_5F : BOOL;
		Pritomn_PowerCP_5H : BOOL;
		PrazdnaPoziciaTopCoveru : BOOL;
	END_STRUCT;
	ControlUnit_typ : 	STRUCT  (*Riadiaci systém pre kamery*)
		Profinet_PLC_INPUTS : ARRAY[0..1]OF USINT;
		Stav_READY : BOOL;
	END_STRUCT;
END_TYPE

(*******************Devlink*****************************)

TYPE
	StrukturaNovehoNazvuAdresara_typ : 	STRUCT
		LINKA : STRING[11]; (*Názov linky PowerCP*)
		PRACOVISKO : STRING[10]; (*ST1,ST2,ST3 .......*)
		ROK : STRING[10]; (*YYYY*)
		DATUM : STRING[10]; (*YYYY_MM_SS*)
	END_STRUCT;
	StrukturaNovehoNazvuSuboru_typ : 	STRUCT
		DATUM : STRING[10]; (*YYYY_MM_DD*)
		CAS : STRING[8]; (*HH_MM_SS*)
		SERIAL : STRING[30]; (*Kód modelu*)
		INDEX : STRING[2]; (*1,2,3 ......*)
		RESULT : STRING[5]; (*PASS alebo FAIL*)
		Pripona : STRING[5]; (*.jpg*)
	END_STRUCT;
END_TYPE

(***************Posielanie fotiek na server**********************)

TYPE
	FTP_Kamery_typ : 	STRUCT
		CMD : FTP_Kamery_CMD_typ;
		INPUTS : FTP_Kamery_INPUTS_typ;
		STATUS : FTP_Kamery_STATUS_typ;
	END_STRUCT;
	FTP_Kamery_CMD_typ : 	STRUCT
		OdosliFotku : BOOL;
		VymazFotku : BOOL;
	END_STRUCT;
	FTP_Kamery_INPUTS_typ : 	STRUCT
		QRkodPowerCP : STRING[30]; (*Master number*)
		Result : STRING[5]; (*PASS alebo FAIL*)
		IndexFotky : STRING[2];
	END_STRUCT;
	FTP_Kamery_STATUS_typ : 	STRUCT
		KomunikaciaUkoncena : BOOL;
		KomunikaciaError : BOOL;
		PopisPoruchy : STRING[300];
		AdresarPrazdny : BOOL;
		VymazanieAdresaraKamery_BUSY : BOOL;
	END_STRUCT;
END_TYPE
```

### Global.var - Global variables
```iecst
(********************************************************************
 * COPYRIGHT -- Microsoft
 ********************************************************************
 * File: Global.var
 * Author: Martin
 * Created: February 11, 2016
 ********************************************************************
 * Global variables of project Zamazat_1
 ********************************************************************)
VAR
	QRkod_PowerCP : STRING[30] := '';
END_VAR
(**********Nastavenie času**************)
VAR
	DTSetTime_0 : DTSetTime;
	DTGetTime_0 : DTGetTime;
END_VAR
(******************Blikače*****************************)
VAR
	Blikac100ms : BOOL;
	Blikac200ms : BOOL;
	Blikac500ms : BOOL;
	Blikac1s : BOOL;
END_VAR
(********************Safety**********************************)
VAR
	Safety : Safety_typ := (0);
END_VAR
(********************Vizualizacia*****************************)
VAR
	Vizu : Vizu_typ;
	P1_Vizu : P1_Vizu_typ;
	P2_Vizu : P2_Vizu_typ;
	P34_Vizu : P34_Vizu_typ;
	FilterVizu_P1 : STRING[300];
	FilterVizu_P2 : STRING[300];
	FilterVizu_P34 : STRING[300];
END_VAR
(**************Remanentné premenné*********)
VAR
	P1_RemPremenne : P1_RemPremenne_typ;
	P2_RemPremenne : P2_RemPremenne_typ;
	P34_RemPremenne : P34_RemPremenne_typ;
	MpRecipeXml_P1 : MpRecipeXml := (0);
	MpRecipeRegPar_P1 : MpRecipeRegPar := (0);
	MpRecipeUI_P1 : MpRecipeUI;
	P1_UlozPremenne : BOOL;
	P1_NacitajPremenne : BOOL;
	MpRecipeXml_P2 : MpRecipeXml := (0);
	MpRecipeRegPar_P2 : MpRecipeRegPar := (0);
	MpRecipeUI_P2 : MpRecipeUI;
	P2_UlozPremenne : BOOL;
	P2_NacitajPremenne : BOOL;
	MpRecipeXml_P34 : MpRecipeXml := (0);
	MpRecipeRegPar_P34 : MpRecipeRegPar := (0);
	MpRecipeUI_P34 : MpRecipeUI;
	P34_UlozPremenne : BOOL;
	P34_NacitajPremenne : BOOL;
END_VAR
(*************Tracebility***********************)
VAR
	TRCB_P1_Vytah_ST1 : KOM_Server_typ;
	TRCB_P1_Srobovanie_ST2 : KOM_Server_typ;
	TRCB_P2_ZakladacTesnenia_ST3 : KOM_Server_typ;
	TRCB_P2_Maticovacka_ST4 : KOM_Server_typ;
	TRCB_P2_Srobovanie_ST5 : KOM_Server_typ;
	TRCB_P2_Zvaranie_ST6 : KOM_Server_typ;
	TRCB_P3_Srobovanie_ST7 : KOM_Server_typ;
	TRCB_P3_LeakageTestA_ST8A : KOM_Server_typ;
	TRCB_P3_LeakageTestB_ST8B : KOM_Server_typ;
	TRCB_P4_Etiketovacka_ST9 : KOM_Server_typ;
	TRCB_P4_Vytah_ST10 : KOM_Server_typ;
	TRCB_P1_Vytah_OpatovnyDopyt : BOOL := FALSE;
	TRCB_P1_Vytah_PaletkaNG : BOOL;
	TRCB_P1_Srobov_OpatovnyDopyt : BOOL;
	TRCB_P1_Srobov_PaletkaNG : BOOL;
	TRCB_P2_ZaklTesn_OpatovnyDopyt : BOOL;
	TRCB_P2_ZaklTesn_PaletkaNG : BOOL;
	TRCB_P2_Maticov_OpatovnyDopyt : BOOL;
	TRCB_P2_Maticov_PaletkaNG : BOOL;
	TRCB_P2_Srobov_OpatovnyDopyt : BOOL;
	TRCB_P2_Srobov_PaletkaNG : BOOL;
	TRCB_P2_Zvaranie_OpatovnyDopyt : BOOL;
	TRCB_P2_Zvaranie_PaletkaNG : BOOL;
	TRCB_P3_Srobov_OpatovnyDopyt : BOOL;
	TRCB_P3_Srobov_PaletkaNG : BOOL;
	TRCB_P3_LeakTestA_OpatovnyDopyt : BOOL;
	TRCB_P3_LeakTestA_PaletkaNG : BOOL;
	TRCB_P3_LeakTestB_OpatovnyDopyt : BOOL;
	TRCB_P3_LeakTestB_PaletkaNG : BOOL;
	TRCB_P4_Etiketov_OpatovnyDopyt : BOOL;
	TRCB_P4_Etiketov_PaletkaNG : BOOL;
	TRCB_P4_Vytah_OpatovnyDopyt : BOOL;
	TRCB_P4_Vytah_PaletkaNG : BOOL;
END_VAR
(*****************Kamery***********************************)
VAR
	CAM2 : CAM2_typ; (*P1_ST1_Vytah - kontrola kusov na paletke*)
	CAM3 : CAM3_typ; (*P1_ST1_Vytah - kontrola QR kódu DPS*)
	CAM4 : CAM4_typ; (*P1_ST1_Vytah - kontrola klipov krytu DPS*)
	CAM5 : CAM5_typ; (*P1_ST1_Vytah - kontrola QR kódu PowerCP*)
	CAM6 : CAM6_typ; (*P1_ST2_StoperSkrutkovania - Kontrola paletky*)
	CAM1 : CAM1_typ; (*P2_ST1_ZaklTesnenia - Kontrola tesnenia a QR kódu Power CP*)
	CAM7 : CAM7_typ; (*P2_ST1_StoperZaklTesnenia - Kontrola Power CP a QR kódu filtra*)
	CAM8 : CAM8_typ; (*P2_ST1_StoperZaklTesnenia - Kontrola spodného QR kódu Power CP*)
	CAM9 : CAM9_typ; (*P2_ST2_StoperMaticovacky - Kontrola paletky*)
	CAM10 : CAM10_typ; (*P2_ST3_StoperSkrutkovania - Kontrola paletky*)
	CAM11 : CAM11_typ; (*P2_ST4_StoperZvarania - Kontrola pravého MV case*)
	CAM12 : CAM12_typ; (*P2_ST4_StoperZvarania - Kontrola lavého MV case a Power CP*)
	CAM17 : CAM17_typ; (*P2_ST1_StoperZaklTesnenia - Kontrola paletky*)
	CAM13 : CAM13_typ; (*P3_ST1_StoperSkrutkovania - Kontrola paletky*)
	CAM14 : CAM14_typ; (*P4_ST3_StoperEtiketovania - kontrola QR kodu na Power CP*)
	CAM15 : CAM15_typ; (*P4_ST3_StoperEtiketovania - kontrola nalepenej etikety*)
	CAM16 : CAM16_typ; (*P4_ST4_Vytah - kontrola paletky*)
	ControlUnit : ControlUnit_typ;
	CAM1_PocetFotiek : USINT := 0;
	CAM2_PocetFotiek : USINT := 0;
	CAM3_PocetFotiek : USINT := 0;
	CAM4_PocetFotiek : USINT := 0;
	CAM5_PocetFotiek : USINT := 0;
	CAM6_PocetFotiek : USINT := 0;
	CAM7_PocetFotiek : USINT := 0;
	CAM8_PocetFotiek : USINT := 0;
	CAM9_PocetFotiek : USINT := 0;
	CAM10_PocetFotiek : USINT := 0;
	CAM11_PocetFotiek : USINT := 0;
	CAM12_PocetFotiek : USINT := 0;
	CAM13_PocetFotiek : USINT := 0;
	CAM14_PocetFotiek : USINT := 0;
	CAM15_PocetFotiek : USINT := 0;
	CAM16_PocetFotiek : USINT := 0;
	CAM17_PocetFotiek : USINT := 0;
END_VAR
(***************Odosielanie fotiek na server**************************)
VAR
	FTP_CAM1 : FTP_Kamery_typ; (*ST3 - zakladanie tesnenia - kontrola tesnenia*)
	FTP_CAM2 : FTP_Kamery_typ; (*ST1 - výtah - kontrola paletky*)
	FTP_CAM4 : FTP_Kamery_typ; (*ST1 - výtah - kontrola krytu DPS modely 4F a 5F*)
	FTP_CAM6 : FTP_Kamery_typ; (*ST2 - srobovanie - kontrola paletky*)
	FTP_CAM9 : FTP_Kamery_typ; (*ST4 - maticovacka - kontrola paletky*)
	FTP_CAM10 : FTP_Kamery_typ; (*ST5 - srobovanie - kontrola paletky*)
	FTP_CAM11 : FTP_Kamery_typ; (*ST6 - zváranie - kontrola Power CP*)
	FTP_CAM12 : FTP_Kamery_typ; (*ST6 - zváranie - kontrola paletky*)
	FTP_CAM15 : FTP_Kamery_typ; (*ST9 - etiketovacka - kontrola etikety*)
	FTP_CAM16 : FTP_Kamery_typ; (*ST10 - vytah - kontrola paletky*)
	FTP_CAM17 : FTP_Kamery_typ; (*ST3 - zakladanie tesnenia - kontrola paletky*)
	OdpojServerFTP : BOOL := FALSE;
	Stav_PripojenieFTP_OK : BOOL := FALSE;
	TypFotky_BMP : BOOL := FALSE;
END_VAR
(******************Premenné linky***************************)
VAR RETAIN
	Paletka : ARRAY[0..30] OF Paletka_typ := [31((0))];
END_VAR
VAR
	Linka : Linka_typ := (0);
	Reports : Reports_typ;
	P1_Pracovisko : P1_Pracovisko_typ := (0);
	P1_Vytah : P1_Vytah_typ := (0);
	SC_P1_Vytah : SequenceControlTyp := (0);
	P1_Dopravniky : P1_Dopravniky_typ := (0);
	SC_P1_Dopravniky : SequenceControlTyp := (0);
	P1_SpodnyStoper : P1_SpodnyStoper_typ := (0);
	SC_P1_SpodnyStoper : SequenceControlTyp := (0);
	P1_StoperSrobovania : P1_StoperSrobovania_typ := (0);
	SC_P1_StoperSrobovania : SequenceControlTyp := (0);
	P1_Srobovanie : P1_Srobovanie_typ := (0);
	SC_P1_Srobovanie : SequenceControlTyp := (0);
	P1_AkumulacnyStoper : P1_AkumulacnyStoper_typ := (0);
	SC_P1_AkumulacnyStoper : SequenceControlTyp := (0);
	P1_Robot : P1_Robot_typ := (0);
	SC_P1_Robot : SequenceControlTyp := (0);
	P2_Pracovisko : P2_Pracovisko_typ := (0);
	P2_Dopravniky : P2_Dopravniky_typ := (0);
	SC_P2_Dopravniky : SequenceControlTyp := (0);
	P2_SpodnyStoper : P2_SpodnyStoper_typ := (0);
	SC_P2_SpodnyStoper : SequenceControlTyp := (0);
	P2_StoperZaklTesnenia : P2_StoperZaklTesnenia_typ;
	SC_P2_StoperZaklTesnenia : SequenceControlTyp;
	P2_ZakladacTesnenia : P2_ZakladacTesnenia_typ;
	SC_P2_ZakladacTesnenia : SequenceControlTyp;
	P2_StoperMaticovacky : P2_StoperMaticovacky_typ;
	SC_P2_StoperMaticovacky : SequenceControlTyp;
	P2_AkumulacnyStoper : P2_AkumulacnyStoper_typ := (0);
	SC_P2_AkumulacnyStoper : SequenceControlTyp := (0);
	P2_StoperSrobovania : P2_StoperSrobovania_typ := (0);
	SC_P2_StoperSrobovania : SequenceControlTyp := (0);
	P2_Srobovanie : P2_Srobovanie_typ := (0);
	SC_P2_Srobovanie : SequenceControlTyp := (0);
	P2_Robot : P2_Robot_typ := (0);
	SC_P2_Robot : SequenceControlTyp := (0);
	P2_StoperZvarania : P2_StoperZvarania_typ := (0);
	SC_P2_StoperZvarania : SequenceControlTyp := (0);
	P2_Zvaranie : P2_Zvaranie_typ;
	SC_P2_Zvaranie : SequenceControlTyp;
	P2_Cistenie : P2_Cistenie_typ;
	SC_P2_Cistenie : SequenceControlTyp;
	P3_Pracovisko : P3_Pracovisko_typ := (0);
	P3_Dopravniky : P3_Dopravniky_typ := (0);
	SC_P3_Dopravniky : SequenceControlTyp := (0);
	P3_SpodnyStoper : P3_SpodnyStoper_typ := (0);
	SC_P3_SpodnyStoper : SequenceControlTyp := (0);
	P3_StoperSrobovania : P3_StoperSrobovania_typ := (0);
	SC_P3_StoperSrobovania : SequenceControlTyp := (0);
	P3_Srobovanie : P3_Srobovanie_typ := (0);
	SC_P3_Srobovanie : SequenceControlTyp := (0);
	P3_HV_Test : P3_HV_Test_typ := (0);
	SC_P3_HV_Test : SequenceControlTyp := (0);
	P3_ZdvizkaPredLeakTestA : P3_ZdvizkaPredLeakTestA_typ := (0);
	SC_P3_ZdvizkaPredLeakTestA : SequenceControlTyp := (0);
	P3_ZdvizkaPredLeakTestB : P3_ZdvizkaPredLeakTestB_typ := (0);
	SC_P3_ZdvizkaPredLeakTestB : SequenceControlTyp := (0);
	P3_LeakageTestA : P3_LeakageTestA_typ;
	SC_P3_LeakageTestA : SequenceControlTyp;
	AteqLeakageTester_A : AteqTester_typ;
	P3_LeakageTestB : P3_LeakageTestB_typ;
	SC_P3_LeakageTestB : SequenceControlTyp;
	AteqLeakageTester_B : AteqTester_typ;
	P3_ZdvizkaZaLeakTestA : P3_ZdvizkaZaLeakTestA_typ := (0);
	SC_P3_ZdvizkaZaLeakTestA : SequenceControlTyp := (0);
	P3_ZdvizkaZaLeakTestB : P3_ZdvizkaZaLeakTestB_typ := (0);
	SC_P3_ZdvizkaZaLeakTestB : SequenceControlTyp := (0);
	P4_Pracovisko : P4_Pracovisko_typ := (0);
	P4_Dopravniky : P4_Dopravniky_typ := (0);
	SC_P4_Dopravniky : SequenceControlTyp := (0);
	P4_SpodnyStoper : P4_SpodnyStoper_typ := (0);
	SC_P4_SpodnyStoper : SequenceControlTyp := (0);
	P4_FunkcnyTestA : P4_FunkcnyTestA_typ;
	SC_P4_FunkcnyTestA : SequenceControlTyp;
	P4_FunkcnyTestB : P4_FunkcnyTestB_typ;
	SC_P4_FunkcnyTestB : SequenceControlTyp;
	P4_ZdvizkaZaFunkcTestA : P4_ZdvizkaZaFunkcTestA_typ := (0);
	SC_P4_ZdvizkaZaFunkcTestA : SequenceControlTyp := (0);
	P4_ZdvizkaZaFunkcTestB : P4_ZdvizkaZaFunkcTestB_typ := (0);
	SC_P4_ZdvizkaZaFunkcTestB : SequenceControlTyp := (0);
	P4_Etiketovacka : P4_Etiketovacka_typ;
	SC_P4_Etiketovacka : SequenceControlTyp;
	P4_Vytah : P4_Vytah_typ;
	SC_P4_Vytah : SequenceControlTyp;
END_VAR
(********************Príznaky********************************)
VAR
	P1_Vytah_KAM_Result_Ignoruj : BOOL;
	P1_Srobov_KAM_Result_OK : BOOL := 0;
	P1_Srobov_KAM_Result_NG : BOOL := 0;
	P1_Srobov_KAM_Result_Ignoruj : BOOL := FALSE;
	P1_Srobov_K30_Result_OFF : BOOL := 0;
	P1_Srobov_M4_Result_OFF : BOOL := 0;
	P1_Srobov_M5_Result_OFF : BOOL := 0;
	P2_ZaklTesn_KAM_Result_Ignoruj : BOOL;
	P2_Maticov_KAM_Result_OK : BOOL;
	P2_Maticov_KAM_Result_NG : BOOL;
	P2_Maticov_KAM_Result_Ignoruj : BOOL;
	P2_Maticov_MaticaM4_Result_OFF : BOOL := FALSE;
	P2_Srobov_KAM_Result_OK : BOOL;
	P2_Srobov_KAM_Result_NG : BOOL;
	P2_Srobov_KAM_Result_Ignoruj : BOOL;
	P2_Srobov_M6_Result_OFF : BOOL := FALSE;
	P2_Srobov_M5_Result_OFF : BOOL := FALSE;
	P2_Srobov_M4_Result_OFF : BOOL := FALSE;
	P2_Zvaranie_KAM_Result_NG : BOOL;
	P2_Zvaranie_KAM_Result_OK : BOOL;
	P3_Srobov_KAM_Result_Ignoruj : BOOL;
	P3_Srobov_KAM_Result_OK : BOOL;
	P3_Srobov_KAM_Result_NG : BOOL;
	P3_Srobov_K40_Result_OFF : BOOL := FALSE;
	P3_Srobov_M5_Result_OFF : BOOL := FALSE;
	P4_Etiketov_KAM_Result_OK : BOOL;
	P4_Etiketov_KAM_Result_NG : BOOL;
	P4_Etiketov_KAM_Result_Ignoruj : BOOL;
	P4_Vytah_KAM_Result_NG : BOOL;
	P4_Vytah_KAM_Result_OK : BOOL;
	P4_Vytah_KAM_Result_Ignoruj : BOOL;
END_VAR
(************Taktime pracovisk****************)
VAR
	P1_Vytah_Taktime : Taktime := (0);
	P1_Skrutkovanie_Taktime : Taktime := (0);
	P2_ZakladanieTesnenia_Taktime : Taktime := (0);
	P2_Maticovacka_Taktime : Taktime := (0);
	P2_Skrutkovanie_Taktime : Taktime := (0);
	P2_Zvaranie_Taktime : Taktime := (0);
	P3_Skrutkovanie_Taktime : Taktime := (0);
	P3_HVtest_Taktime : Taktime := (0);
	P3_LeakageTestA_Taktime : Taktime := (0);
	P3_LeakageTestB_Taktime : Taktime := (0);
	P4_FinalTestA_Taktime : Taktime := (0);
	P4_FinalTestB_Taktime : Taktime := (0);
	P4_Etiketovanie_Taktime : Taktime := (0);
	P4_Vytah_Taktime : Taktime := (0);
END_VAR
```

### Package Logical/Libraries - Global libraries

### Library Logical/Libraries/IecCheck (IEC)
Depends on: sys_lib, AsBrStr

#### IecCheck.fun - Exported functions and function blocks
```iecst
FUNCTION CheckDivSint : SINT (* Check divisor for SINT division *)
	VAR_INPUT
		divisor : SINT;
	END_VAR
END_FUNCTION

FUNCTION CheckDivUsint : USINT (* Check divisor for USINT division *)
	VAR_INPUT
		divisor : USINT;
	END_VAR
END_FUNCTION

FUNCTION CheckDivInt : INT (* Check divisor for INT division *)
	VAR_INPUT
		divisor : INT;
	END_VAR
END_FUNCTION

FUNCTION CheckDivUint : UINT (* Check divisor for UINT division *)
	VAR_INPUT
		divisor : UINT;
	END_VAR
END_FUNCTION

FUNCTION CheckDivDint : DINT (* Check divisor for DINT division *)
	VAR_INPUT
		divisor : DINT;
	END_VAR
END_FUNCTION

FUNCTION CheckDivUdint : UDINT (* Check divisor for UDINT division *)
	VAR_INPUT
		divisor : UDINT;
	END_VAR
END_FUNCTION

FUNCTION CheckDivReal : REAL (* Check divisor for REAL division *)
	VAR_INPUT
		divisor : REAL;
	END_VAR
END_FUNCTION

FUNCTION CheckDivLReal : LREAL (* Check divisor for LREAL division, not available for SG3 and SGC *)
	VAR_INPUT
		divisor : LREAL;
	END_VAR
END_FUNCTION

FUNCTION CheckBounds : DINT (* Check range for array access *)
	VAR_INPUT
		index : DINT;
		lower : DINT;
		upper : DINT;
	END_VAR
END_FUNCTION

FUNCTION CheckRange : DINT (* Check range for enumeration *)
	VAR_INPUT
		value : DINT;
		lower : DINT;
		upper : DINT;
	END_VAR
END_FUNCTION

FUNCTION CheckSignedSubrange : DINT (* Check range for subrange of signed data types *)
	VAR_INPUT
		value : DINT;
		lower : DINT;
		upper : DINT;
	END_VAR
END_FUNCTION

FUNCTION CheckUnsignedSubrange : UDINT (* Check range for subrange of unsigned data types *)
	VAR_INPUT
		value : UDINT;
		lower : UDINT;
		upper : UDINT;
	END_VAR
END_FUNCTION

FUNCTION CheckReadAccess : UDINT (* Check address when reading dynamic variables *)
	VAR_INPUT
		address : UDINT;
	END_VAR
END_FUNCTION

FUNCTION CheckWriteAccess : UDINT (* Check address when writing dynamic variables *)
	VAR_INPUT
		address : UDINT;
	END_VAR
END_FUNCTION

FUNCTION MakeEntry : UDINT (* Makes an entry (log book entry) in the error log book *)
	VAR
		taskname : STRING[30];
		group : USINT;
		status_name : UINT;
		out_text : STRING[80];
	END_VAR
	VAR_INPUT
		number : UINT;
		index : DINT;
		text : STRING[50];
	END_VAR
END_FUNCTION
```

#### IecCheck.st - Implementation file
```iecst
(* Check divisor for SINT division *)
FUNCTION CheckDivSint
	IF divisor=0 THEN
		CheckDivSint:=1;
		MakeEntry(55555,divisor,'CheckDivSint');
	ELSE
		CheckDivSint:=divisor;
	END_IF
END_FUNCTION

(* Check divisor for USINT division *)
FUNCTION CheckDivUsint
	IF divisor=0 THEN
		CheckDivUsint:=1;
		MakeEntry(55555,divisor,'CheckDivUsint');
	ELSE
		CheckDivUsint:=divisor;
	END_IF
END_FUNCTION

(* Check divisor for INT division *)
FUNCTION CheckDivInt
	IF divisor=0 THEN
		CheckDivInt:=1;
		MakeEntry(55555,divisor,'CheckDivInt');
	ELSE
		CheckDivInt:=divisor;
	END_IF
END_FUNCTION

(* Check divisor for UINT division *)
FUNCTION CheckDivUint
	IF divisor=0 THEN
		CheckDivUint:=1;
		MakeEntry(55555,divisor,'CheckDivUint');
	ELSE
		CheckDivUint:=divisor;
	END_IF
END_FUNCTION

(* Check divisor for DINT division *)
FUNCTION CheckDivDint
	IF divisor=0 THEN
		CheckDivDint:=1;
		MakeEntry(55555,divisor,'CheckDivDint');
	ELSE
		CheckDivDint:=divisor;
	END_IF
END_FUNCTION

(* Check divisor for UDINT division *)
FUNCTION CheckDivUdint
	IF divisor=0 THEN
		CheckDivUdint:=1;
		MakeEntry(55555,divisor,'CheckDivUdint');
	ELSE
		CheckDivUdint:=divisor;
	END_IF
END_FUNCTION

(* Check divisor for REAL division *)
FUNCTION CheckDivReal
	IF divisor=0 THEN
		CheckDivReal:=1;
		MakeEntry(55555,0,'CheckDivReal');
	ELSE
		CheckDivReal:=divisor;
	END_IF
END_FUNCTION

(* Check divisor for LREAL division *)
FUNCTION CheckDivLReal
	IF divisor=0 THEN
		CheckDivLReal:=1;
		MakeEntry(55555,0,'CheckDivLReal');
	ELSE
		CheckDivLReal:=divisor;
	END_IF
END_FUNCTION

(* Check range for array access *)
FUNCTION CheckBounds
	IF index < lower THEN
		CheckBounds := lower;
		MakeEntry(55555,index,'CheckBounds');
	ELSIF index > upper THEN
		CheckBounds := upper;
		MakeEntry(55555,index,'CheckBounds');
	ELSE
		CheckBounds := index;
	END_IF
END_FUNCTION

(* Check range for enumeration *)
FUNCTION CheckRange
	IF value < lower THEN
		CheckRange := lower;
		MakeEntry(55555,value,'CheckRange');
	ELSIF value > upper THEN
		CheckRange := upper;
		MakeEntry(55555,value,'CheckRange');
	ELSE
		CheckRange := value;
	END_IF
END_FUNCTION

(* Check range for subrange of signed data types *)
FUNCTION CheckSignedSubrange
	IF value < lower THEN
		CheckSignedSubrange := lower;
		MakeEntry(55555,value,'CheckSignedSubrange');
	ELSIF value > upper THEN
		CheckSignedSubrange := upper;
		MakeEntry(55555,value,'CheckSignedSubrange');
	ELSE
		CheckSignedSubrange := value;
	END_IF
END_FUNCTION

(* Check range for subrange of unsigned data types *)
FUNCTION CheckUnsignedSubrange
	IF value < lower THEN
		CheckUnsignedSubrange := lower;
		MakeEntry(55555,value,'CheckUnsignedSubrange');
	ELSIF value > upper THEN
		CheckUnsignedSubrange := upper;
		MakeEntry(55555,value,'CheckUnsignedSubrange');
	ELSE
		CheckUnsignedSubrange := value;
	END_IF
END_FUNCTION

(* Check address when reading dynamic variables *)
FUNCTION CheckReadAccess
	IF address=0 THEN
		(* TODO: Insert an appropriate code, see AutomationStudio help for further information *)
		MakeEntry(55555,address,'Read from NULL');
	END_IF

	CheckReadAccess:=0;
END_FUNCTION

(* Check address when writing dynamic variables *)
FUNCTION CheckWriteAccess
	IF address=0 THEN
		(* TODO: Insert an appropriate code, see AutomationStudio help for further information *)
		MakeEntry(55555,address,'Write to NULL');
	END_IF

	CheckWriteAccess:=0;
END_FUNCTION

(* Makes an entry (log book entry) in the error log book *)
FUNCTION MakeEntry
		status_name := ST_name(0,ADR(taskname),ADR(group));

		brsstrcpy(ADR(out_text),ADR(text));
		brsstrcat(ADR(out_text),ADR(' > in task > '));
  		brsstrcat(ADR(out_text),ADR(taskname));
		MakeEntry := ADR(out_text);
		ERRxfatal(number,index,ADR(out_text));
END_FUNCTION
```

### Library Logical/Libraries/SC (IEC)

#### Types.typ - Exported data types
```iecst
TYPE
	SequenceControlTyp : 	STRUCT
		StepName : STRING[255];
		Step : UINT;
		Switch1 : BOOL;
		Switch2 : BOOL;
		Switch3 : BOOL;
		ResetStep : BOOL;
		LastStep : BOOL;
		IdleTime : TON;
		AlarmTime : TON;
	END_STRUCT;
END_TYPE
```

#### SC.fun - Exported functions and function blocks
```iecst
FUNCTION SequenceControl : BOOL
	VAR_IN_OUT
		SC : SequenceControlTyp;
	END_VAR
END_FUNCTION
```

#### SequenceControl.st
```iecst
(* TODO: Add your comment here *)
FUNCTION SequenceControl

	IF SC.ResetStep THEN
		brsmemset(ADR(SC.StepName),0,SIZEOF(SC.StepName));
		SC.Switch1:= FALSE;
		SC.Switch2:= FALSE;
		SC.Switch3:= FALSE;
		SC.IdleTime.IN:= FALSE;
		SC.AlarmTime.IN:= FALSE;
		SC.ResetStep:= FALSE;
	END_IF

	IF SC.LastStep THEN
		brsmemset(ADR(SC.StepName),0,SIZEOF(SC.StepName));
		SC.Switch1:= FALSE;
		SC.Switch2:= FALSE;
		SC.Switch3:= FALSE;
		SC.IdleTime.IN:= FALSE;
		SC.AlarmTime.IN:= FALSE;
		SC.Step:= 0;
		SC.LastStep:= FALSE;
	END_IF

	//Volanie časovačov//
	SC.AlarmTime();
	SC.IdleTime();

END_FUNCTION
```

### Library Logical/Libraries/Banner (IEC)

#### Types.typ - Exported data types
```iecst
TYPE
	Banner_IN_typ : 	STRUCT
		CervenaLED_ON : BOOL;
		ZelenaLED_ON : BOOL;
		ModraLED_ON : BOOL;
		OranzovaLED_ON : BOOL;
		ZltaLED_ON : BOOL;
		CyanLED_ON : BOOL;
		ModraRotujucaLED_ON : BOOL;
		Blikac100ms : BOOL;
	END_STRUCT;
	Banner_OUT_typ : 	STRUCT
		Stlaceny : BOOL;
	END_STRUCT;
END_TYPE
```

#### Banner.fun - Exported functions and function blocks
```iecst
{REDUND_ERROR} FUNCTION_BLOCK BannerIOlink (*Banner na IO linku*) (*$GROUP=User,$CAT=User,$GROUPICON=User.png,$CATICON=User.png*)
	VAR_INPUT
		Mapping_IN : {REDUND_UNREPLICABLE} ARRAY[0..15] OF USINT;
		IN : {REDUND_UNREPLICABLE} Banner_IN_typ;
	END_VAR
	VAR_OUTPUT
		Mapping_OUT : ARRAY[0..15] OF USINT;
		OUT : Banner_OUT_typ;
	END_VAR
	VAR
		Step : USINT;
		zzEdge00000 : BOOL;
	END_VAR
END_FUNCTION_BLOCK
```

#### BannerIOlink.st
```iecst
(* Banner na IO linku *)
FUNCTION_BLOCK BannerIOlink

	//*****************Banner stlačený********************//
	OUT.Stlaceny:= Mapping_IN[1].0;

	//*******************Banner zmena farieb******************//
	IF IN.CervenaLED_ON THEN
		Mapping_OUT[2]:= 161;
		Mapping_OUT[3]:= 161;
		Mapping_OUT[4]:= 161;
		Mapping_OUT[5]:= 161;
		Mapping_OUT[6]:= 161;
		Mapping_OUT[7]:= 161;
		Mapping_OUT[8]:= 161;
		Mapping_OUT[9]:= 161;
	ELSIF IN.ZelenaLED_ON THEN
		Mapping_OUT[2]:= 160;
		Mapping_OUT[3]:= 160;
		Mapping_OUT[4]:= 160;
		Mapping_OUT[5]:= 160;
		Mapping_OUT[6]:= 160;
		Mapping_OUT[7]:= 160;
		Mapping_OUT[8]:= 160;
		Mapping_OUT[9]:= 160;
	ELSIF IN.ModraLED_ON THEN
		Mapping_OUT[2]:= 169;
		Mapping_OUT[3]:= 169;
		Mapping_OUT[4]:= 169;
		Mapping_OUT[5]:= 169;
		Mapping_OUT[6]:= 169;
		Mapping_OUT[7]:= 169;
		Mapping_OUT[8]:= 169;
		Mapping_OUT[9]:= 169;
	ELSIF IN.OranzovaLED_ON THEN
		Mapping_OUT[2]:= 162;
		Mapping_OUT[3]:= 162;
		Mapping_OUT[4]:= 162;
		Mapping_OUT[5]:= 162;
		Mapping_OUT[6]:= 162;
		Mapping_OUT[7]:= 162;
		Mapping_OUT[8]:= 162;
		Mapping_OUT[9]:= 162;
	ELSIF IN.ZltaLED_ON THEN
		Mapping_OUT[2]:= 164;
		Mapping_OUT[3]:= 164;
		Mapping_OUT[4]:= 164;
		Mapping_OUT[5]:= 164;
		Mapping_OUT[6]:= 164;
		Mapping_OUT[7]:= 164;
		Mapping_OUT[8]:= 164;
		Mapping_OUT[9]:= 164;
	ELSIF IN.CyanLED_ON THEN
		Mapping_OUT[2]:= 167;
		Mapping_OUT[3]:= 167;
		Mapping_OUT[4]:= 167;
		Mapping_OUT[5]:= 167;
		Mapping_OUT[6]:= 167;
		Mapping_OUT[7]:= 167;
		Mapping_OUT[8]:= 167;
		Mapping_OUT[9]:= 167;
	ELSIF IN.ModraRotujucaLED_ON THEN
		IF EDGEPOS(IN.Blikac100ms)THEN
			IF Mapping_OUT[5] = 160 THEN
				Mapping_OUT[2]:= 160;
				Mapping_OUT[6]:= 160;
				Mapping_OUT[3]:= 160;
				Mapping_OUT[7]:= 160;
				Mapping_OUT[4]:= 169;
				Mapping_OUT[8]:= 169;
				Mapping_OUT[5]:= 169;
				Mapping_OUT[9]:= 169;
			ELSIF Mapping_OUT[2] = 160 THEN
				Mapping_OUT[2]:= 169;
				Mapping_OUT[6]:= 169;
				Mapping_OUT[3]:= 160;
				Mapping_OUT[7]:= 160;
				Mapping_OUT[4]:= 160;
				Mapping_OUT[8]:= 160;
				Mapping_OUT[5]:= 169;
				Mapping_OUT[9]:= 169;
			ELSIF Mapping_OUT[8] = 160 THEN
				Mapping_OUT[2]:= 169;
				Mapping_OUT[6]:= 169;
				Mapping_OUT[3]:= 169;
				Mapping_OUT[7]:= 169;
				Mapping_OUT[4]:= 160;
				Mapping_OUT[8]:= 160;
				Mapping_OUT[5]:= 160;
				Mapping_OUT[9]:= 160;
			ELSIF Mapping_OUT[9] = 160 THEN
				Mapping_OUT[2]:= 160;
				Mapping_OUT[6]:= 160;
				Mapping_OUT[3]:= 169;
				Mapping_OUT[7]:= 169;
				Mapping_OUT[4]:= 169;
				Mapping_OUT[8]:= 169;
				Mapping_OUT[5]:= 160;
				Mapping_OUT[9]:= 160;
			ELSE
				Mapping_OUT[5]:= 160;
			END_IF
		END_IF
	ELSE
		Mapping_OUT[2]:= 0;
		Mapping_OUT[3]:= 0;
		Mapping_OUT[4]:= 0;
		Mapping_OUT[5]:= 0;
		Mapping_OUT[6]:= 0;
		Mapping_OUT[7]:= 0;
		Mapping_OUT[8]:= 0;
		Mapping_OUT[9]:= 0;
	END_IF

END_FUNCTION_BLOCK
```

### Library Logical/Libraries/RFID (IEC, version 3.10.0) - A new source library

#### RFID.typ - Exported data types
```iecst
(********************************************************************
 * COPYRIGHT -- Bernecker + Rainer
 ********************************************************************
 * Library: RFID
 * File: RFID.typ
 * Author: houx
 * Created: March 25, 2009
 ********************************************************************
 * Data types of library RFID
 ********************************************************************)

TYPE
	Info : 	STRUCT
		ID : UDINT;
		Type : UDINT;
		StackLevel : UDINT;
	END_STRUCT;
	status : 	STRUCT
		GetUsbList : UINT;
		GetUsbNode : UINT;
		ReleaseBuffer : UINT;
		XOPEN : UINT;
		WRITE : UINT;
		READ : UINT;
		GetBuffer : UINT;
		RoBuffer : UINT;
	END_STRUCT;
	usbDevice : 	STRUCT
		vendorID : UDINT;
		productId : UDINT;
		bcdDevice : UDINT;
	END_STRUCT;
END_TYPE

(**)
```

#### RFID.var - Exported constants
```iecst
(********************************************************************
 * COPYRIGHT -- Bernecker + Rainer
 ********************************************************************
 * Library: RFID
 * File: RFID.var
 * Author: houx
 * Created: March 25, 2009
 ********************************************************************
 * Constants of library RFID
 ********************************************************************)
VAR CONSTANT
	REG1 : USINT := 1;
	REG2 : USINT := 2;
	REG4 : USINT := 4;
	REG5 : USINT := 5;
	REG6 : USINT := 6;
	REG8 : USINT := 8;
	REG9 : USINT := 9;
	REG11 : USINT := 11;
	REG14 : USINT := 14;
	REG13 : USINT := 13;
	REG12 : USINT := 12;
	REG10 : USINT := 10;
	REG7 : USINT := 7;
	REG15 : USINT := 15;
	REG16 : USINT := 16;
	REG19 : USINT := 19;
	REG18 : USINT := 18;
	REG17 : USINT := 17;
	REG20 : USINT := 20;
	REG25 : USINT := 25;
	REG26 : USINT := 26;
	REG28 : USINT := 28;
	READ : USINT := 2;
	WRITE : USINT := 1;
	REG30 : USINT := 30;
	REG33 : USINT := 33;
	CLOSE : USINT := 100;
	REG32 : USINT := 32;
	REG31 : USINT := 31;
	SEARCHTP : USINT := 1;
	SEARCHTPLIST : USINT := 0;
	REG29 : USINT := 29;
	REG27 : USINT := 27;
	STACKWRITE : USINT := 5;
	TRANSPONDER_VENDOR_ID : UINT := 1659;
	TYPEREAD : USINT := 2;
	TRANSPONDER_PRODUCT_ID : UINT := 8963;
	TYPEWRITE : USINT := 1;
	TRANSPONDER_BCD : UINT := 768;
	STACKREAD : USINT := 6;
	REG24 : USINT := 24;
	RW : USINT := 1;
	REG23 : USINT := 23;
	REG22 : USINT := 22;
	REG21 : USINT := 21;
	OPEN : USINT := 0;
	IDWRITE : USINT := 3;
	IDREAD : USINT := 4;
	rfidError_lock_wrongType : UDINT := 41;
	rfidError_password_wrongType : UDINT := 61;
	rfidError_stacklevel_failed : UDINT := 23;
	rfidError_unlock_failed : UDINT := 52;
	rfidError_unlock_wrongType : UDINT := 51;
	rfidError_tag_failed : UDINT := 21;
	rfidError_crc_failed : USINT := 31;
	rfidError_id_failed : UDINT := 22;
	rfidError_write_failed : UDINT := 83;
	rfidError_write_wrongRegNr : UDINT := 82;
	rfidError_write_wrongType : UDINT := 81;
	rfidError_read_wrongRegNr : UDINT := 72;
	rfidError_read_wrongType : UDINT := 71;
	rfidError_rf_failed : UDINT := 11;
	rfidError_read_failed : UDINT := 73;
	rfidError_password_failed : UDINT := 62;
	rfidError_lock_failed : UDINT := 42;
	DATAREAD : USINT := 3;
	REG3 : USINT := 3;
END_VAR
```

#### RFID.fun - Exported functions and function blocks
```iecst
FUNCTION_BLOCK TP_Init (*TODO: Add your comment here*)
	VAR_INPUT
		Enable : BOOL; (*Add your parameter comment*)
	END_VAR
	VAR_OUTPUT
		Ident : ARRAY[0..10] OF UDINT;
		Error : BOOL;
		ErrorID : UDINT;
		Busy : BOOL;
		Done : BOOL;
	END_VAR
	VAR
		StepInit : USINT;
		USBNodeListGetFuB : UsbNodeListGet;
		status : status;
		usbNodeList : ARRAY[0..31] OF UDINT;
		i : UINT;
		USBNodeGetFuB : UsbNodeGet;
		usbDevice : ARRAY[0..10] OF usbNode_typ;
		StringDevice : ARRAY[0..10] OF STRING[30];
	END_VAR
END_FUNCTION_BLOCK
(********************************************************************
 * COPYRIGHT -- Bernecker + Rainer
 ********************************************************************
 * Library: RFID
 * File: RFID.fun
 * Author: houx
 * Created: March 25, 2009
 ********************************************************************
 * Functions and function blocks of library RFID
 ********************************************************************)

FUNCTION_BLOCK TP_Info (*TODO: Add your comment here*)
	VAR_INPUT
		Enable : BOOL; (*Add your parameter comment*)
		Ident : UDINT;
	END_VAR
	VAR_OUTPUT
		Busy : BOOL;
		Done : BOOL;
		Error : BOOL;
		ErrorID : UDINT;
		Info : Info;
	END_VAR
	VAR
		Stepstatus : USINT;
		WriteData : ARRAY[0..255] OF USINT;
		FrameWriteStruct : FRM_write;
		status : status;
		FrameReadStruct : FRM_read;
		ReadBuffer : UDINT;
		ReadBufferLength : UINT;
		ReadData : ARRAY[0..255] OF USINT;
		FrameReleaseBufferStruct : FRM_rbuf;
		ID : ARRAY[0..9] OF USINT;
		StackLevel : ARRAY[0..1] OF USINT;
		KeyType : ARRAY[0..3] OF USINT;
		AN : ARRAY[0..2] OF USINT;
		sendbuffer : UDINT;
		FrameGetBufferStruct : FRM_gbuf;
		sendbufferlength : UINT;
		FrameReleaseOutputBufferStruct : FRM_robuf;
		FrameXOpenStruct : FRM_xopen;
	END_VAR
END_FUNCTION_BLOCK

FUNCTION_BLOCK TP_Unlock (*TODO: Add your comment here*)
	VAR_INPUT
		Enable : BOOL; (*Add your parameter comment*)
		Ident : UDINT;
		Data : UDINT;
	END_VAR
	VAR_OUTPUT
		Busy : BOOL;
		Error : BOOL;
		ErrorID : UDINT;
		Done : BOOL;
	END_VAR
	VAR
		StepType : USINT;
		WriteData : ARRAY[0..255] OF USINT;
		FrameWriteStruct : FRM_write;
		status : status;
		FrameReadStruct : FRM_read;
		ReadBuffer : UDINT;
		ReadBufferLength : UINT;
		ReadData : ARRAY[0..255] OF USINT;
		FrameReleaseBufferStruct : FRM_rbuf;
		string1 : STRING[20];
		string2 : STRING[10];
		CMD : UDINT;
		StepWrite : USINT;
		ERROR : ARRAY[0..2] OF USINT;
		AN : ARRAY[0..2] OF USINT;
		FrameGetBufferStruct : FRM_gbuf;
		sendbuffer : UDINT;
		sendbufferlength : UINT;
		FrameReleaseOutputBufferStruct : FRM_robuf;
		FrameXOpenStruct : FRM_xopen;
		TypeOK : BOOL;
	END_VAR
END_FUNCTION_BLOCK

FUNCTION_BLOCK TP_Lock (*TODO: Add your comment here*)
	VAR_INPUT
		Enable : BOOL; (*Add your parameter comment*)
		Ident : UDINT;
	END_VAR
	VAR_OUTPUT
		Busy : BOOL;
		ErrorID : UDINT;
		Error : BOOL;
		Done : BOOL;
	END_VAR
	VAR
		WriteData : ARRAY[0..255] OF USINT;
		FrameWriteStruct : FRM_write;
		status : status;
		FrameReadStruct : FRM_read;
		ReadBuffer : UDINT;
		ReadData : ARRAY[0..255] OF USINT;
		ReadBufferLength : UINT;
		FrameReleaseBufferStruct : FRM_rbuf;
		StepLOCK : USINT;
		AN : ARRAY[0..2] OF USINT;
		ERROR : ARRAY[0..2] OF USINT;
		TypeOK : BOOL;
		StepType : USINT;
		FrameGetBufferStruct : FRM_gbuf;
		sendbufferlength : UINT;
		sendbuffer : UDINT;
		FrameReleaseOutputBufferStruct : FRM_robuf;
		FrameXOpenStruct : FRM_xopen;
	END_VAR
END_FUNCTION_BLOCK

FUNCTION_BLOCK TP_PWProtect (*TODO: Add your comment here*)
	VAR_INPUT
		Enable : BOOL; (*Add your parameter comment*)
		Ident : UDINT;
		Data : UDINT;
	END_VAR
	VAR_OUTPUT
		Busy : BOOL;
		Error : BOOL;
		ErrorID : UDINT;
		Done : BOOL;
	END_VAR
	VAR
		TypeOK : BOOL;
		StepType : USINT;
		WriteData : ARRAY[0..255] OF USINT;
		FrameWriteStruct : FRM_write;
		status : status;
		FrameReadStruct : FRM_read;
		ReadBuffer : UDINT;
		ReadBufferLength : UINT;
		ReadData : ARRAY[0..255] OF USINT;
		FrameReleaseBufferStruct : FRM_rbuf;
		string1 : STRING[20];
		string2 : STRING[20];
		CMD : UDINT;
		StepWrite : USINT;
		AN : ARRAY[0..2] OF USINT;
		ERROR : ARRAY[0..2] OF USINT;
		FrameGetBufferStruct : FRM_gbuf;
		sendbuffer : UDINT;
		sendbufferlength : UINT;
		FrameReleaseOutputBufferStruct : FRM_robuf;
		FrameXOpenStruct : FRM_xopen;
	END_VAR
END_FUNCTION_BLOCK

FUNCTION_BLOCK TP_OnOff (*TODO: Add your comment here*)
	VAR_INPUT
		Enable : BOOL; (*Add your parameter comment*)
		Ident : UDINT;
		Mode : BOOL;
	END_VAR
	VAR_OUTPUT
		Error : BOOL;
		ErrorID : UDINT;
		Busy : BOOL;
		Done : BOOL;
	END_VAR
	VAR
		StepOnOff : USINT;
		WriteData : ARRAY[0..255] OF USINT;
		FrameWriteStruct : FRM_write;
		status : status;
		FrameReadStruct : FRM_read;
		ReadBuffer : UDINT;
		ReadBufferLength : UINT;
		ReadData : ARRAY[0..255] OF USINT;
		FrameReleaseOutputBufferStruct : FRM_robuf;
		AN : ARRAY[0..2] OF USINT;
		FrameGetBufferStruct : FRM_gbuf;
		sendbuffer : UDINT;
		sendbufferlength : UINT;
		FrameReleaseBufferStruct : FRM_rbuf;
		FrameXOpenStruct : FRM_xopen;
		FRM_close_0 : FRM_close;
	END_VAR
END_FUNCTION_BLOCK

FUNCTION_BLOCK TP_Crc (*TODO: Add your comment here*)
	VAR_INPUT
		Enable : BOOL; (*Add your parameter comment*)
		Ident : UDINT;
		Mode : BOOL;
	END_VAR
	VAR_OUTPUT
		Error : BOOL;
		ErrorID : UDINT;
		Busy : BOOL;
		Done : BOOL;
	END_VAR
	VAR
		WriteData : ARRAY[0..255] OF USINT;
		FrameWriteStruct : FRM_write;
		FrameReadStruct : FRM_read;
		ReadBuffer : UDINT;
		ReadData : ARRAY[0..255] OF USINT;
		ReadBufferLength : UINT;
		FrameReleaseBufferStruct : FRM_rbuf;
		status : status;
		StepCRC : USINT;
		AN : ARRAY[0..2] OF USINT;
		FrameGetBufferStruct : FRM_gbuf;
		sendbuffer : UDINT;
		sendbufferlength : UINT;
		FrameReleaseOutputBufferStruct : FRM_robuf;
		FrameXOpenStruct : FRM_xopen;
		FRM_close_0 : FRM_close;
	END_VAR
END_FUNCTION_BLOCK

FUNCTION_BLOCK TP_Write (*TODO: Add your comment here*)
	VAR_INPUT
		Enable : BOOL; (*Add your parameter comment*)
		RegNr : USINT;
		Data : UDINT;
		Ident : UDINT;
	END_VAR
	VAR_OUTPUT
		Busy : BOOL;
		Error : BOOL;
		ErrorID : UDINT;
		Done : BOOL;
	END_VAR
	VAR
		CMD : UDINT;
		WriteData : ARRAY[0..255] OF USINT;
		StepWrite : USINT;
		FrameWriteStruct : FRM_write;
		status : status;
		CommandReady : BOOL;
		ReadBuffer : UDINT;
		FrameReleaseBufferStruct : FRM_rbuf;
		ReadBufferLength : UINT;
		FrameReadStruct : FRM_read;
		ReadData : ARRAY[0..255] OF USINT;
		string1 : STRING[30];
		string2 : STRING[30];
		StepType : USINT;
		TypeOK : BOOL;
		string3 : STRING[10];
		AN : ARRAY[0..2] OF USINT;
		ERROR : ARRAY[0..2] OF USINT;
		KeyType : ARRAY[0..3] OF USINT;
		FrameGetBufferStruct : FRM_gbuf;
		sendbuffer : UDINT;
		sendbufferlength : UINT;
		FrameReleaseOutputBufferStruct : FRM_robuf;
		FrameXOpenStruct : FRM_xopen;
	END_VAR
END_FUNCTION_BLOCK

FUNCTION_BLOCK TP_Read (*TODO: Add your comment here*)
	VAR_INPUT
		Enable : BOOL; (*Add your parameter comment*)
		RegNr : USINT;
		Ident : UDINT;
	END_VAR
	VAR_OUTPUT
		Done : BOOL;
		Error : BOOL;
		ErrorID : UDINT;
		Busy : BOOL;
		Data : UDINT;
	END_VAR
	VAR
		CommandReady : BOOL;
		WriteData : ARRAY[0..255] OF USINT;
		status : status;
		ReadBuffer : UDINT;
		ReadBufferLength : UINT;
		ReadData : ARRAY[0..255] OF USINT;
		FrameReadStruct : FRM_read;
		data : ARRAY[0..19] OF USINT;
		FrameReleaseBufferStruct : FRM_rbuf;
		FrameWriteStruct : FRM_write;
		TypeOK : BOOL;
		StepType : USINT;
		KeyType : ARRAY[0..3] OF USINT;
		AN : ARRAY[0..2] OF USINT;
		ERROR : ARRAY[0..2] OF USINT;
		FrameGetBufferStruct : FRM_gbuf;
		sendbuffer : UDINT;
		sendbufferlength : UINT;
		FrameReleaseOutputBufferStruct : FRM_robuf;
		FrameXOpenStruct : FRM_xopen;
		StepREAD : USINT;
	END_VAR
END_FUNCTION_BLOCK
```

#### TP_Init.st
```iecst
(********************************************************************
 * COPYRIGHT -- Bernecker + Rainer
 ********************************************************************
 * Library: RFID
 * File: TP_Init.st
 * Author: houx
 * Created: March 25, 2009
 *****************************************************************
FuB: 			TP_Init
*****************************************************************
Discription:
	USB Interface:	This FuB find the Transponder Reader(USB) in the Target and read out the Interface Ident.
								Interface Ident ist required for all other FuBs in RFID Library.
								This FuB can work without any transponder in the range of Reader.
	serial Interface:	This FuB is not used to find a serial interface transponder reader
Parameter:
	Input:
		Enable(BOOL)	: The function block is only executed when enable is <> 0
	Output:
		Error(BOOL)		: Error = 0 (No Error) Error = 1(see ErrorID)
		ErrorID(UDINT)	: Number and Description in Error Table
		Busy(BOOL)		: Fub working on
		Ident(UDINT)	: Interface ID
		Done(BOOL)		: success, if TRUE
Author:	Xiaoguang Hou
		B&R Eggelsberg

History: 	V1.00.0 - 02 Sep 2008 first create
				V3.00.0 - 25 Mar 2009  update for serial interface transponder reader and created under AS3.0

*****************************************************************

 ********************************************************************
 * Implementation of library RFID
 ********************************************************************)

FUNCTION_BLOCK TP_Init

(*------------------------------------------------------	Start	---------------------------------------------------------*)
IF Enable = TRUE THEN
	IF (Done = FALSE) AND (Error = FALSE) THEN
		Busy	:=	TRUE;
		CASE StepInit OF
	(*	------------------------------------------------	search usb device	---------------------------------------------*)
			SEARCHTPLIST :
				USBNodeListGetFuB(enable := TRUE,pBuffer := ADR(usbNodeList),bufferSize := SIZEOF(usbNodeList));
				status.GetUsbList				:=USBNodeListGetFuB.status;
				IF status.GetUsbList = 0  THEN
					StepInit					:=SEARCHTP;
					USBNodeListGetFuB.enable 	:= FALSE;
				END_IF
	(*	------------------------------------------------	if Error ?show ErrorID	----------------------------------------------------*)
				IF (status.GetUsbList <> 0) AND (status.GetUsbList <> 65535) THEN
					StepInit 	:= SEARCHTPLIST;
					Error		:= TRUE;
					Busy		:= FALSE;
					ErrorID		:= status.GetUsbList;
				END_IF
	(*	----------------------------------------------- usb device identizification , a Transponder ? get the deviceID----------------------*)
			SEARCHTP:
				USBNodeGetFuB(enable := TRUE,nodeId := usbNodeList[i],pBuffer := ADR(usbDevice[i]),bufferSize :=256 (*SIZEOF(usbDevice)*));
				status.GetUsbNode := USBNodeGetFuB.status;
				IF  status.GetUsbNode = 0 THEN
					IF	(usbDevice[i].vendorId = TRANSPONDER_VENDOR_ID) AND (usbDevice[i].productId = TRANSPONDER_PRODUCT_ID) AND (usbDevice[i].bcdDevice = TRANSPONDER_BCD) THEN
						strcpy(ADR(StringDevice[i]),ADR(usbDevice[i].ifName));
						Ident[i]				:= ADR(StringDevice[i]);
						Done                    := TRUE;
						Busy                    := FALSE;
						USBNodeGetFuB.enable 	:= FALSE;
						i						:= i+1;
						IF i= USBNodeListGetFuB.listNodes THEN
							i           	        := 0;
							StepInit				:= SEARCHTPLIST;
						END_IF
					ELSE
						i						:= i+1;
					END_IF
				ELSIF status.GetUsbNode = 65535 THEN
					StepInit				:=SEARCHTP;
				ELSE
					StepInit :=  SEARCHTPLIST;
					Error 	 :=  TRUE;
					Busy     :=  FALSE;
					ErrorID  :=  status.GetUsbNode;
				END_IF
		END_CASE
	END_IF
	(*	------------------------------------------------	Not Enable, set parameters FALSE	----------------------------------------------------*)
ELSE
	Busy	:=	FALSE;
	Error	:=	FALSE;
	Done	:=	FALSE;
	ErrorID	:=	FALSE;
END_IF
(*	------------------------------------------------	end	----------------------------------------------------*)
END_FUNCTION_BLOCK
```

#### TP_Info.st
```iecst
(********************************************************************
 * COPYRIGHT -- Bernecker + Rainer
 ********************************************************************
 * Library: RFID
 * File: TP_Info.st
 * Author: houx
 * Created: March 25, 2009
*****************************************************************
FuB: 			TP_Info
;*****************************************************************
Discription:
	This FuB can be used to output the Transponder Type, the stack lever and HW/SW	versions.
	This Fub can only work, if any Transponder in the range of Reader.
	Type			: 4150 R/W or 4102 R
	Stack level		: stack level in transponder memory
	HW/SW version	:	guarantees that your application software is being operated with the correct readers.
Parameter:
			Input: 		Enable(BOOL)	:	The function block is only executed when enable is <> 0
				   			Ident(UDINT)	:	Interface Ident from TP_Init.
			Output: 	Error(BOOL)		:	Error = 0 (No Error) Error = 1(see ErrorID)
							ErrorID(UDINT)	:	Number and Description in Error Table
							Busy(BOOL)		:	if TRUE , Fub working on.
							Done(BOOL)		:	if TRUE, success
							Info(Info)		:	Structure with Type, ID and Stacklevel.
Author:				Xiaoguang Hou
							B&R Eggelsberg
;History:	V1.00.0 - 02 Sep 2008 : first create
				V3.00.0 - 25 Mar 2009 : update for serial interface transponder and created under AS3.0
 ********************************************************************
 * Implementation of library RFID
 ********************************************************************)

FUNCTION_BLOCK TP_Info
(*--------------------------------------	start	----------------------------*)
IF (Enable = 1) THEN
	IF ((Done = 0) AND (Error = 0)) THEN
		Busy	:=	TRUE;
		CASE Stepstatus OF
(*	------------------------------------------------	open the interface, get the internal Ident	----------------------------------------------------*)
			OPEN:
				FrameXOpenStruct(enable := 1,device := Ident);
				status.XOPEN 			:= FrameXOpenStruct.status;
				IF (status.XOPEN = 0) THEN
					Stepstatus          := TYPEWRITE ;
					FrameXOpenStruct.enable := FALSE;
				ELSE
					Stepstatus          := OPEN ;
					Error               := TRUE;
					ErrorID             := status.XOPEN;
					Busy                := 0;
				END_IF
			TYPEWRITE:
				memset(ADR(WriteData),0,SIZEOF(WriteData));
				strcpy(ADR(WriteData),ADR('tag,0,0,#crc$R$L'));
				FrameGetBufferStruct(enable:= 1, ident:= FrameXOpenStruct.ident);
				sendbuffer					:= FrameGetBufferStruct.buffer;
				sendbufferlength		:= FrameGetBufferStruct.buflng;
				status.GetBuffer		:= FrameGetBufferStruct.status;
				IF	(status.GetBuffer = 0)	THEN
					memcpy(sendbuffer,ADR(WriteData),sendbufferlength);
					FrameWriteStruct(enable := 1, ident := FrameXOpenStruct.ident, buffer := sendbuffer,buflng := strlen(ADR(WriteData)));
					status.WRITE 			:=	FrameWriteStruct.status;
				  	IF (status.WRITE <> 0) THEN
						FrameReleaseOutputBufferStruct(enable:=1,ident:=FrameXOpenStruct.ident,buffer:=sendbuffer,buflng:=strlen(ADR(WriteData)) );
						status.RoBuffer			:= FrameReleaseOutputBufferStruct.status;
					ELSE
				    	FrameGetBufferStruct.enable	:= 0;
						FrameWriteStruct.enable := 0;
						FrameReleaseOutputBufferStruct.enable := 0;
						Stepstatus              :=	TYPEREAD;
					END_IF
				ELSE
					ErrorID 	:= status.GetBuffer;
					Error   	:= 1;
					Busy    	:= 0;
					FrameGetBufferStruct.enable	:= 0;
					Stepstatus	:= OPEN;
				END_IF
			TYPEREAD:
				FrameReadStruct(enable:=1,ident:=FrameXOpenStruct.ident);
				ReadBuffer       	:=	FrameReadStruct.buffer;
				ReadBufferLength	:=	FrameReadStruct.buflng;
				status.READ      	:=	FrameReadStruct.status;
				IF  (status.READ = 0) THEN
					memset(ADR(ReadData),0,SIZEOF(ReadData));
					memcpy(ADR(ReadData),ReadBuffer,ReadBufferLength);                   (* copy read data into read buffer *)
					FrameReadStruct.enable	:= 0;
			        FrameReleaseBufferStruct(enable:=1, ident:=FrameXOpenStruct.ident, buffer:=ReadBuffer,buflng:=ReadBufferLength);        (* release read buffer *)
			        status.ReleaseBuffer	:=FrameReleaseBufferStruct.status;
			        IF (status.ReleaseBuffer=0) THEN
				        FrameReleaseBufferStruct.enable:=0;
						AN[0]		 :=	ReadData[0];
						AN[1]		 := ReadData[1];
						AN[2]		 := ReadData[2];
						IF	(memcmp(ADR(AN),ADR('ack'),3) = 0)	THEN
							memset(ADR(KeyType),0,SIZEOF(KeyType));
							KeyType[0]   	 := ReadData[6];
							KeyType[1] 	 := ReadData[7];
							KeyType[2] 	 := ReadData[8];
							KeyType[3] 	 := ReadData[9];
							IF (memcmp(ADR(KeyType),ADR('4150'),4) = 0) THEN
								Info.Type	:=	ADR(KeyType);
								Stepstatus	:=	IDWRITE;
							ELSIF	(memcmp(ADR(KeyType),ADR('4102'),4) = 0) THEN
								Info.Type	:=	ADR(KeyType);
								Stepstatus	:=	IDWRITE;
							ELSE
								Stepstatus	:= OPEN;
								ErrorID	:=	rfidError_tag_failed; (* unknow type of transponder *)
								Error   :=	1;
								Busy    :=	0;
							END_IF
						ELSIF	(memcmp(ADR(AN),ADR('nak'),3) = 0)	THEN
							Stepstatus	:= OPEN;
							ErrorID	:=	rfidError_tag_failed; (* negativ answer *)
							Error   :=	1;
							Busy    :=	0;
						ELSE
							Stepstatus	:= OPEN;
							ErrorID	:=	rfidError_tag_failed; (* unknow answer *)
							Error   :=	1;
							Busy    :=	0;
						END_IF
					ELSE
						Stepstatus	:=	OPEN;
						Error     	:=	1;
						ErrorID   	:=	status.ReleaseBuffer;
						Busy      	:=	0;
					END_IF
				ELSE
					memset(ADR(ReadData),0,SIZEOF(ReadData));
				END_IF
			IDWRITE:
				memset(ADR(WriteData),0,SIZEOF(WriteData));
				strcpy(ADR(WriteData),ADR('id,0,#crc$R$L'));
				FrameGetBufferStruct(enable:= 1, ident:= FrameXOpenStruct.ident);
				sendbuffer				    := FrameGetBufferStruct.buffer;
				sendbufferlength		:= FrameGetBufferStruct.buflng;
				status.GetBuffer		:= FrameGetBufferStruct.status;
				IF	(status.GetBuffer = 0)	THEN
					memcpy(sendbuffer,ADR(WriteData),sendbufferlength);
					FrameWriteStruct(enable := 1, ident := FrameXOpenStruct.ident, buffer := sendbuffer,buflng := strlen(ADR(WriteData)));
					status.WRITE 			:=	FrameWriteStruct.status;

			        IF (status.WRITE <> 0) THEN
						FrameReleaseOutputBufferStruct(enable:=1,ident:=FrameXOpenStruct.ident,buffer:=sendbuffer,buflng:= strlen(ADR(WriteData)));
						status.RoBuffer			:= FrameReleaseOutputBufferStruct.status;
						IF	(status.RoBuffer <> 0)	THEN
							ErrorID	:= status.RoBuffer;
						END_IF
					ELSE
			        	FrameWriteStruct.enable := 0;
						FrameGetBufferStruct.enable	:= 0;
						FrameReleaseOutputBufferStruct.enable := 0;
						Stepstatus              :=	IDREAD;
					END_IF
				ELSE
					ErrorID 	:= status.GetBuffer;
					Error   	:= 1;
					Busy    	:= 0;
					Stepstatus	:= OPEN;
					FrameGetBufferStruct.enable	:= 0;
				END_IF

			IDREAD:
				FrameReadStruct(enable:=1,ident:=FrameXOpenStruct.ident);
				ReadBuffer       	:=	FrameReadStruct.buffer;
				ReadBufferLength	:=	FrameReadStruct.buflng;
				status.READ      	:=	FrameReadStruct.status;
				IF  (status.READ = 0) THEN
					memset(ADR(ReadData),0,SIZEOF(ReadData));
					memcpy(ADR(ReadData),ReadBuffer,ReadBufferLength);                   (* copy read data into read buffer *)
					FrameReadStruct.enable	:=	0;
			        FrameReleaseBufferStruct(enable:=1, ident:=FrameXOpenStruct.ident, buffer:=ReadBuffer,buflng:=ReadBufferLength);        (* release read buffer *)
			        status.ReleaseBuffer	:=	FrameReleaseBufferStruct.status;
			        IF (status.ReleaseBuffer=0) THEN
				        FrameReleaseBufferStruct.enable	:=	0;
				        AN[0]	:= ReadData[0];
						AN[1]	:= ReadData[1];
						AN[2]	:= ReadData[2];
				        IF	(memcmp(ADR(AN),ADR('ack'),3) = 0) THEN
				        	memset(ADR(ID),0,SIZEOF(ID));
							ID[0] 	 	:=	ReadData[6];
							ID[1] 	 	:=	ReadData[7];
							ID[2] 	 	:=	ReadData[8];
							ID[3] 	 	:=	ReadData[9];
							ID[4] 	 	:=	ReadData[11];
							ID[5] 	 	:=	ReadData[12];
							ID[6] 	 	:=	ReadData[13];
							ID[7] 	 	:=	ReadData[14];
							Info.ID   	:=	ADR(ID);
							Stepstatus  :=	STACKWRITE;
						ELSE
							Stepstatus	:= OPEN;
							Error     	:= 1;
							ErrorID   	:= rfidError_id_failed;	(* negativ answer by ask for ID *)
							Busy      	:= 0;
						END_IF
					ELSE
						Stepstatus	:= OPEN;
						Error     	:= 1;
						ErrorID   	:= status.ReleaseBuffer;
						Busy      	:= 0;
					END_IF
				ELSE
					memset(ADR(ReadData),0,SIZEOF(ReadData));
				END_IF
			STACKWRITE:
				memset(ADR(WriteData),0,SIZEOF(WriteData));
				strcpy(ADR(WriteData),ADR('stack,0,#crc$R$L'),);
				FrameGetBufferStruct(enable:= 1, ident:= FrameXOpenStruct.ident);
				sendbuffer				:= FrameGetBufferStruct.buffer;
				sendbufferlength		:= FrameGetBufferStruct.buflng;
				status.GetBuffer		:= FrameGetBufferStruct.status;
				IF	(status.GetBuffer = 0)	THEN
					memcpy(sendbuffer,ADR(WriteData),sendbufferlength);
					FrameWriteStruct(enable := 1, ident := FrameXOpenStruct.ident, buffer := sendbuffer,buflng := strlen(ADR(WriteData)));
					status.WRITE 		:=	FrameWriteStruct.status;
			        Stepstatus          :=	STACKREAD;
			        IF (status.WRITE <> 0) THEN
						FrameReleaseOutputBufferStruct(enable:=1,ident:=FrameXOpenStruct.ident,buffer:=sendbuffer,buflng:= strlen(ADR(WriteData)));
						status.RoBuffer			:= FrameReleaseOutputBufferStruct.status;
						IF	(status.RoBuffer <> 0)	THEN
							ErrorID	:= status.RoBuffer;
						END_IF
					END_IF
					FrameWriteStruct.enable :=	0;
					FrameGetBufferStruct.enable	:= 0;
					FrameReleaseOutputBufferStruct.enable := 0;
				ELSE
					ErrorID 	:= status.GetBuffer;
					Error   	:= 1;
					Busy    	:= 0;
					Stepstatus	:= OPEN;
					FrameGetBufferStruct.enable	:= 0;
				END_IF
			STACKREAD:
				FrameReadStruct(enable:=1,ident:=FrameXOpenStruct.ident);
				ReadBuffer       	:=	FrameReadStruct.buffer;
				ReadBufferLength	:=	FrameReadStruct.buflng;
				status.READ      	:=	FrameReadStruct.status;
				IF  (status.READ = 0) THEN
					memset(ADR(ReadData),0,SIZEOF(ReadData));
					memcpy(ADR(ReadData),ReadBuffer,ReadBufferLength);                   (* copy read data into read buffer *)
					FrameReadStruct.enable	:=	0;
			        FrameReleaseBufferStruct(enable:=1, ident:=FrameXOpenStruct.ident, buffer:=ReadBuffer,buflng:=ReadBufferLength);        (* release read buffer *)
			        status.ReleaseBuffer	:=	FrameReleaseBufferStruct.status;
			        IF (status.ReleaseBuffer = 0) THEN
				        FrameReleaseBufferStruct.enable	:=	0;
				        AN[0]	:= ReadData[0];
						AN[1]	:= ReadData[1];
						AN[2]	:= ReadData[2];
				        IF	(memcmp(ADR(AN),ADR('ack'),3) = 0) THEN
							memset(ADR(StackLevel),0,SIZEOF(StackLevel));
							StackLevel[0] 	  :=	ReadData[6];
							StackLevel[1] 	  :=	ReadData[7];
							Info.StackLevel :=	ADR(StackLevel);
							Stepstatus		  :=	OPEN;
							Done			  :=	1;
							Busy			  :=	0;
						ELSE
							Stepstatus	:=	OPEN;
							Error     	:=	1;
							ErrorID   	:=	rfidError_stacklevel_failed;
							Busy      	:=	0;
						END_IF
					ELSE
						Stepstatus	:=	OPEN;
						Error     	:=	1;
						ErrorID   	:=	status.ReleaseBuffer;
						Busy      	:=	0;
					END_IF
				ELSE
					memset(ADR(ReadData),0,SIZEOF(ReadData));
				END_IF
		END_CASE
	END_IF
ELSE
	Busy    := 0;
	Error   := 0;
	ErrorID := 0;
	Done    := 0;
END_IF
END_FUNCTION_BLOCK
```
